LIN {X 0,Y 272.995,Z 1069.366,A -85,B 0,C 180,E1 12162.479,E2 12162.479} C_VEL
LIN {X 0,Y 273.086,Z 1073.952,A -85,B 0,C 180,E1 12158.633,E2 12158.633} C_VEL
LIN {X 0,Y 273.548,Z 1076.686,A -85,B 0,C 180,E1 12155.032,E2 12155.032} C_VEL
LIN {X 0,Y 273.964,Z 1077.76,A -85,B 0,C 180,E1 12151.673,E2 12151.673} C_VEL
LIN {X 0,Y 274.031,Z 1077.444,A -85,B 0,C 180,E1 12148.536,E2 12148.536} C_VEL
LIN {X 0,Y 273.725,Z 1075.691,A -85,B 0,C 180,E1 12145.18,E2 12145.18} C_VEL
LIN {X 0,Y 273.314,Z 1072.175,A -85,B 0,C 180,E1 12141.585,E2 12141.585} C_VEL
LIN {X 0,Y 273.199,Z 1066.916,A -85,B 0,C 180,E1 12137.959,E2 12137.959} C_VEL
LIN {X 0,Y 273.666,Z 1059.821,A -85,B 0,C 180,E1 12134.313,E2 12134.313} C_VEL
LIN {X 0,Y 274.877,Z 1050.701,A -85,B 0,C 180,E1 12130.669,E2 12130.669} C_VEL
LIN {X 0,Y 276.832,Z 1040.026,A -85,B 0,C 180,E1 12127.265,E2 12127.265} C_VEL
LIN {X 0,Y 279.412,Z 1027.805,A -85,B 0,C 180,E1 12124.114,E2 12124.114} C_VEL
LIN {X 0,Y 282.522,Z 1014.014,A -85,B 0,C 180,E1 12121.228,E2 12121.228} C_VEL
LIN {X 0,Y 285.89,Z 999.163,A -85,B 0,C 180,E1 12118.71,E2 12118.71} C_VEL
LIN {X 0,Y 289.318,Z 983.345,A -85,B 0,C 180,E1 12116.549,E2 12116.549} C_VEL
LIN {X 0,Y 292.639,Z 966.616,A -85,B 0,C 180,E1 12114.73,E2 12114.73} C_VEL
LIN {X 0,Y 295.712,Z 948.926,A -85,B 0,C 180,E1 12113.239,E2 12113.239} C_VEL
LIN {X 0,Y 298.36,Z 930.328,A -85,B 0,C 180,E1 12112.082,E2 12112.082} C_VEL
LIN {X 0,Y 300.252,Z 911.657,A -85,B 0,C 180,E1 12111.268,E2 12111.268} C_VEL
LIN {X 0,Y 301.36,Z 889.6,A -85,B 0,C 180,E1 12110.665,E2 12110.665} C_VEL
LIN {X 0,Y 306.573,Z 751.848,A -85,B 0,C 180,E1 12107.521,E2 12107.521} C_VEL
LIN {X 0,Y 305.583,Z 740.205,A -85,B 0,C 180,E1 12106.999,E2 12106.999} C_VEL
LIN {X 0,Y 309.064,Z 717.613,A -85,B 0,C 180,E1 12105.112,E2 12105.112} C_VEL
LIN {X 0,Y 307.717,Z 708.174,A -85,B 0,C 180,E1 12102.748,E2 12102.748} C_VEL
LIN {X 0,Y 307.382,Z 698.126,A -85,B 0,C 180,E1 12099.852,E2 12099.852} C_VEL
LIN {X 0,Y 308.086,Z 690.154,A -85,B 0,C 180,E1 12097.025,E2 12097.025} C_VEL
LIN {X 0,Y 309.031,Z 686.401,A -85,B 0,C 180,E1 12095.504,E2 12095.504} C_VEL
LIN {X 0,Y 308.64,Z 688.001,A -85,B 0,C 180,E1 12091.921,E2 12091.921} C_VEL
LIN {X 0,Y 309.095,Z 689.328,A -85,B 0,C 180,E1 12090.092,E2 12090.092} C_VEL
LIN {X 0,Y 310.043,Z 693.073,A -85,B 0,C 180,E1 12087.462,E2 12087.462} C_VEL
LIN {X 0,Y 311.425,Z 698.192,A -85,B 0,C 180,E1 12084.871,E2 12084.871} C_VEL
LIN {X 0,Y 312.988,Z 704.764,A -85,B 0,C 180,E1 12082.343,E2 12082.343} C_VEL
LIN {X 0,Y 314.593,Z 713.54,A -85,B 0,C 180,E1 12079.688,E2 12079.688} C_VEL
LIN {X 0,Y 315.406,Z 720.749,A -85,B 0,C 180,E1 12077.908,E2 12077.908} C_VEL
LIN {X 0,Y 311.769,Z 746.11,A -85,B 0,C 180,E1 12074.225,E2 12074.225} C_VEL
LIN {X 0,Y 312.167,Z 749.946,A -85,B 0,C 180,E1 12073.919,E2 12073.919} C_VEL
LIN {X 0,Y 302.573,Z 860.757,A -85,B 0,C 180,E1 12070.273,E2 12070.273} C_VEL
LIN {X 0,Y 301.167,Z 887.675,A -85,B 0,C 180,E1 12069.157,E2 12069.157} C_VEL
LIN {X 0,Y 299.803,Z 903.792,A -85,B 0,C 180,E1 12068.148,E2 12068.148} C_VEL
LIN {X 0,Y 297.855,Z 918.992,A -85,B 0,C 180,E1 12066.844,E2 12066.844} C_VEL
LIN {X 0,Y 295.433,Z 933.273,A -85,B 0,C 180,E1 12065.243,E2 12065.243} C_VEL
LIN {X 0,Y 292.379,Z 947.73,A -85,B 0,C 180,E1 12063.136,E2 12063.136} C_VEL
LIN {X 0,Y 289.471,Z 959.226,A -85,B 0,C 180,E1 12060.989,E2 12060.989} C_VEL
LIN {X 0,Y 286.549,Z 969.342,A -85,B 0,C 180,E1 12058.6,E2 12058.6} C_VEL
LIN {X 0,Y 283.732,Z 978.089,A -85,B 0,C 180,E1 12055.958,E2 12055.958} C_VEL
LIN {X 0,Y 281.077,Z 985.57,A -85,B 0,C 180,E1 12052.97,E2 12052.97} C_VEL
LIN {X 0,Y 278.881,Z 991.049,A -85,B 0,C 180,E1 12049.881,E2 12049.881} C_VEL
LIN {X 0,Y 277.157,Z 994.834,A -85,B 0,C 180,E1 12046.65,E2 12046.65} C_VEL
LIN {X 0,Y 275.923,Z 996.716,A -85,B 0,C 180,E1 12043.365,E2 12043.365} C_VEL
LIN {X 0,Y 275.168,Z 996.843,A -85,B 0,C 180,E1 12040.028,E2 12040.028} C_VEL
LIN {X 0,Y 274.817,Z 995.053,A -85,B 0,C 180,E1 12036.635,E2 12036.635} C_VEL
LIN {X 0,Y 274.858,Z 991.649,A -85,B 0,C 180,E1 12033.42,E2 12033.42} C_VEL
LIN {X 0,Y 275.278,Z 986.292,A -85,B 0,C 180,E1 12030.158,E2 12030.158} C_VEL
LIN {X 0,Y 276.066,Z 979.37,A -85,B 0,C 180,E1 12027.093,E2 12027.093} C_VEL
LIN {X 0,Y 277.27,Z 970.164,A -85,B 0,C 180,E1 12023.999,E2 12023.999} C_VEL
LIN {X 0,Y 278.662,Z 960.149,A -85,B 0,C 180,E1 12021.367,E2 12021.367} C_VEL
LIN {X 0,Y 280.353,Z 947.978,A -85,B 0,C 180,E1 12018.81,E2 12018.81} C_VEL
LIN {X 0,Y 282.105,Z 934.37,A -85,B 0,C 180,E1 12016.56,E2 12016.56} C_VEL
LIN {X 0,Y 283.657,Z 920.721,A -85,B 0,C 180,E1 12014.757,E2 12014.757} C_VEL
LIN {X 0,Y 285.152,Z 904.969,A -85,B 0,C 180,E1 12013.138,E2 12013.138} C_VEL
LIN {X 0,Y 286.275,Z 889.331,A -85,B 0,C 180,E1 12011.932,E2 12011.932} C_VEL
LIN {X 0,Y 287.078,Z 871.902,A -85,B 0,C 180,E1 12010.982,E2 12010.982} C_VEL
LIN {X 0,Y 288.495,Z 824.298,A -85,B 0,C 180,E1 12009.46,E2 12009.46} C_VEL
LIN {X 0,Y 292.505,Z 735.615,A -85,B 0,C 180,E1 12006.795,E2 12006.795} C_VEL
LIN {X 0,Y 291.348,Z 726.273,A -85,B 0,C 180,E1 12006.299,E2 12006.299} C_VEL
LIN {X 0,Y 293.227,Z 697.722,A -85,B 0,C 180,E1 12002.258,E2 12002.258} C_VEL
LIN {X 0,Y 288.187,Z 679.048,A -85,B 0,C 180,E1 11998.834,E2 11998.834} C_VEL
LIN {X 0,Y 285.826,Z 671.112,A -85,B 0,C 180,E1 11997.219,E2 11997.219} C_VEL
LIN {X 0,Y 285.73,Z 671.591,A -85,B 0,C 180,E1 11996.832,E2 11996.832} C_VEL
LIN {X 0,Y 289.394,Z 684.621,A -85,B 0,C 180,E1 11992.981,E2 11992.981} C_VEL
LIN {X 0,Y 292.427,Z 697.104,A -85,B 0,C 180,E1 11989.63,E2 11989.63} C_VEL
LIN {X 0,Y 296.094,Z 705.518,A -85,B 0,C 180,E1 11988.815,E2 11988.815} C_VEL
LIN {X 0,Y 302.336,Z 742.558,A -85,B 0,C 180,E1 11986.947,E2 11986.947} C_VEL
LIN {X 0,Y 297.857,Z 856.262,A -85,B 0,C 180,E1 11984.229,E2 11984.229} C_VEL
LIN {X 0,Y 296.8,Z 873.568,A -85,B 0,C 180,E1 11983.479,E2 11983.479} C_VEL
LIN {X 0,Y 295.19,Z 890.075,A -85,B 0,C 180,E1 11982.421,E2 11982.421} C_VEL
LIN {X 0,Y 293.048,Z 906.282,A -85,B 0,C 180,E1 11981.016,E2 11981.016} C_VEL
LIN {X 0,Y 290.554,Z 921.277,A -85,B 0,C 180,E1 11979.308,E2 11979.308} C_VEL
LIN {X 0,Y 287.726,Z 935.883,A -85,B 0,C 180,E1 11977.187,E2 11977.187} C_VEL
LIN {X 0,Y 284.947,Z 948.755,A -85,B 0,C 180,E1 11974.831,E2 11974.831} C_VEL
LIN {X 0,Y 282.29,Z 960.021,A -85,B 0,C 180,E1 11972.233,E2 11972.233} C_VEL
LIN {X 0,Y 279.893,Z 969.883,A -85,B 0,C 180,E1 11969.386,E2 11969.386} C_VEL
LIN {X 0,Y 277.876,Z 978.33,A -85,B 0,C 180,E1 11966.287,E2 11966.287} C_VEL
LIN {X 0,Y 276.311,Z 985.211,A -85,B 0,C 180,E1 11962.933,E2 11962.933} C_VEL
LIN {X 0,Y 275.28,Z 990.531,A -85,B 0,C 180,E1 11959.325,E2 11959.325} C_VEL
LIN {X 0,Y 274.824,Z 993.823,A -85,B 0,C 180,E1 11955.892,E2 11955.892} C_VEL
LIN {X 0,Y 274.806,Z 995.381,A -85,B 0,C 180,E1 11952.798,E2 11952.798} C_VEL
LIN {X 0,Y 273.962,Z 995.9,A -85,B 0,C 180,E1 11951.19,E2 11951.19} C_VEL
LIN {X 0,Y 269.946,Z 996.336,A -85,B 0,C 180,E1 11948.118,E2 11948.118} C_VEL
LIN {X 0,Y 268.383,Z 995.852,A -85,B 0,C 180,E1 11946.127,E2 11946.127} C_VEL
LIN {X 0,Y 268.434,Z 995.457,A -85,B 0,C 180,E1 11945.418,E2 11945.418} C_VEL
LIN {X 0,Y 270.205,Z 992.308,A -85,B 0,C 180,E1 11941.727,E2 11941.727} C_VEL
LIN {X 0,Y 272.718,Z 987.361,A -85,B 0,C 180,E1 11938.134,E2 11938.134} C_VEL
LIN {X 0,Y 275.825,Z 980.766,A -85,B 0,C 180,E1 11934.805,E2 11934.805} C_VEL
LIN {X 0,Y 279.405,Z 972.721,A -85,B 0,C 180,E1 11931.751,E2 11931.751} C_VEL
LIN {X 0,Y 283.302,Z 963.298,A -85,B 0,C 180,E1 11928.971,E2 11928.971} C_VEL
LIN {X 0,Y 287.374,Z 952.502,A -85,B 0,C 180,E1 11926.457,E2 11926.457} C_VEL
LIN {X 0,Y 291.479,Z 940.225,A -85,B 0,C 180,E1 11924.199,E2 11924.199} C_VEL
LIN {X 0,Y 295.51,Z 926.416,A -85,B 0,C 180,E1 11922.185,E2 11922.185} C_VEL
LIN {X 0,Y 299.136,Z 911.731,A -85,B 0,C 180,E1 11920.5,E2 11920.5} C_VEL
LIN {X 0,Y 302.219,Z 896.085,A -85,B 0,C 180,E1 11919.121,E2 11919.121} C_VEL
LIN {X 0,Y 304.672,Z 879.206,A -85,B 0,C 180,E1 11918.018,E2 11918.018} C_VEL
LIN {X 0,Y 306.304,Z 861.93,A -85,B 0,C 180,E1 11917.234,E2 11917.234} C_VEL
LIN {X 0,Y 308.486,Z 821.252,A -85,B 0,C 180,E1 11916.181,E2 11916.181} C_VEL
LIN {X 0,Y 312.469,Z 748.774,A -85,B 0,C 180,E1 11914.471,E2 11914.471} C_VEL
LIN {X 0,Y 308.914,Z 728.999,A -85,B 0,C 180,E1 11913.024,E2 11913.024} C_VEL
LIN {X 0,Y 301.266,Z 715.082,A -85,B 0,C 180,E1 11910.738,E2 11910.738} C_VEL
LIN {X 0,Y 293.815,Z 703.135,A -85,B 0,C 180,E1 11908.286,E2 11908.286} C_VEL
LIN {X 0,Y 291.034,Z 698.461,A -85,B 0,C 180,E1 11907.19,E2 11907.19} C_VEL
LIN {X 0,Y 288.191,Z 689.335,A -85,B 0,C 180,E1 11903.163,E2 11903.163} C_VEL
LIN {X 0,Y 285.796,Z 682.579,A -85,B 0,C 180,E1 11899.625,E2 11899.625} C_VEL
LIN {X 0,Y 283.743,Z 676.858,A -85,B 0,C 180,E1 11896.164,E2 11896.164} C_VEL
LIN {X 0,Y 282.053,Z 672.747,A -85,B 0,C 180,E1 11893.114,E2 11893.114} C_VEL
LIN {X 0,Y 280.668,Z 669.223,A -85,B 0,C 180,E1 11890.053,E2 11890.053} C_VEL
LIN {X 0,Y 279.067,Z 665.356,A -85,B 0,C 180,E1 11885.758,E2 11885.758} C_VEL
LIN {X 0,Y 277.614,Z 661.831,A -85,B 0,C 180,E1 11878.762,E2 11878.762} C_VEL
LIN {X 0,Y 277.53,Z 661.462,A -85,B 0,C 180,E1 11874.211,E2 11874.211} C_VEL
LIN {X 0,Y 277.897,Z 662.139,A -85,B 0,C 180,E1 11870.343,E2 11870.343} C_VEL
LIN {X 0,Y 280.251,Z 666.587,A -85,B 0,C 180,E1 11862.776,E2 11862.776} C_VEL
LIN {X 0,Y 282.567,Z 671.568,A -85,B 0,C 180,E1 11858.19,E2 11858.19} C_VEL
LIN {X 0,Y 284.65,Z 676.264,A -85,B 0,C 180,E1 11854.848,E2 11854.848} C_VEL
LIN {X 0,Y 286.664,Z 680.778,A -85,B 0,C 180,E1 11852.136,E2 11852.136} C_VEL
LIN {X 0,Y 289.552,Z 687.256,A -85,B 0,C 180,E1 11848.804,E2 11848.804} C_VEL
LIN {X 0,Y 293.265,Z 696.674,A -85,B 0,C 180,E1 11844.817,E2 11844.817} C_VEL
LIN {X 0,Y 296.357,Z 704.96,A -85,B 0,C 180,E1 11841.934,E2 11841.934} C_VEL
LIN {X 0,Y 304.493,Z 718.116,A -85,B 0,C 180,E1 11839.384,E2 11839.384} C_VEL
LIN {X 0,Y 311.329,Z 730.667,A -85,B 0,C 180,E1 11837.403,E2 11837.403} C_VEL
LIN {X 0,Y 313.145,Z 757.234,A -85,B 0,C 180,E1 11836.102,E2 11836.102} C_VEL
LIN {X 0,Y 305.231,Z 903.639,A -85,B 0,C 180,E1 11832.685,E2 11832.685} C_VEL
LIN {X 0,Y 303.045,Z 922.451,A -85,B 0,C 180,E1 11831.974,E2 11831.974} C_VEL
LIN {X 0,Y 300.035,Z 939.917,A -85,B 0,C 180,E1 11831.033,E2 11831.033} C_VEL
LIN {X 0,Y 296.257,Z 957.297,A -85,B 0,C 180,E1 11829.758,E2 11829.758} C_VEL
LIN {X 0,Y 291.833,Z 974.657,A -85,B 0,C 180,E1 11828.075,E2 11828.075} C_VEL
LIN {X 0,Y 287.145,Z 990.928,A -85,B 0,C 180,E1 11826.048,E2 11826.048} C_VEL
LIN {X 0,Y 282.513,Z 1005.741,A -85,B 0,C 180,E1 11823.726,E2 11823.726} C_VEL
LIN {X 0,Y 277.892,Z 1019.902,A -85,B 0,C 180,E1 11820.965,E2 11820.965} C_VEL
LIN {X 0,Y 273.727,Z 1032.637,A -85,B 0,C 180,E1 11817.875,E2 11817.875} C_VEL
LIN {X 0,Y 270.199,Z 1043.975,A -85,B 0,C 180,E1 11814.452,E2 11814.452} C_VEL
LIN {X 0,Y 267.526,Z 1053.664,A -85,B 0,C 180,E1 11810.796,E2 11810.796} C_VEL
LIN {X 0,Y 265.79,Z 1061.928,A -85,B 0,C 180,E1 11806.837,E2 11806.837} C_VEL
LIN {X 0,Y 265.04,Z 1068.271,A -85,B 0,C 180,E1 11802.86,E2 11802.86} C_VEL
LIN {X 0,Y 265.11,Z 1072.865,A -85,B 0,C 180,E1 11798.838,E2 11798.838} C_VEL
LIN {X 0,Y 265.587,Z 1075.513,A -85,B 0,C 180,E1 11795.183,E2 11795.183} C_VEL
LIN {X 0,Y 266.044,Z 1076.575,A -85,B 0,C 180,E1 11791.722,E2 11791.722} C_VEL
LIN {X 0,Y 266.121,Z 1076.205,A -85,B 0,C 180,E1 11788.492,E2 11788.492} C_VEL
LIN {X 0,Y 265.786,Z 1074.385,A -85,B 0,C 180,E1 11785.036,E2 11785.036} C_VEL
LIN {X 0,Y 265.354,Z 1070.79,A -85,B 0,C 180,E1 11781.331,E2 11781.331} C_VEL
LIN {X 0,Y 265.258,Z 1065.444,A -85,B 0,C 180,E1 11777.592,E2 11777.592} C_VEL
LIN {X 0,Y 265.794,Z 1058.252,A -85,B 0,C 180,E1 11773.836,E2 11773.836} C_VEL
LIN {X 0,Y 267.02,Z 1049.627,A -85,B 0,C 180,E1 11770.305,E2 11770.305} C_VEL
LIN {X 0,Y 269.075,Z 1038.942,A -85,B 0,C 180,E1 11766.803,E2 11766.803} C_VEL
LIN {X 0,Y 271.781,Z 1026.722,A -85,B 0,C 180,E1 11763.566,E2 11763.566} C_VEL
LIN {X 0,Y 275.034,Z 1012.929,A -85,B 0,C 180,E1 11760.607,E2 11760.607} C_VEL
LIN {X 0,Y 278.545,Z 998.068,A -85,B 0,C 180,E1 11758.03,E2 11758.03} C_VEL
LIN {X 0,Y 282.111,Z 982.224,A -85,B 0,C 180,E1 11755.822,E2 11755.822} C_VEL
LIN {X 0,Y 285.56,Z 965.436,A -85,B 0,C 180,E1 11753.967,E2 11753.967} C_VEL
LIN {X 0,Y 288.748,Z 947.603,A -85,B 0,C 180,E1 11752.45,E2 11752.45} C_VEL
LIN {X 0,Y 291.428,Z 929.253,A -85,B 0,C 180,E1 11751.296,E2 11751.296} C_VEL
LIN {X 0,Y 293.355,Z 910.609,A -85,B 0,C 180,E1 11750.475,E2 11750.475} C_VEL
LIN {X 0,Y 294.515,Z 887.782,A -85,B 0,C 180,E1 11749.847,E2 11749.847} C_VEL
LIN {X 0,Y 300.007,Z 753.248,A -85,B 0,C 180,E1 11746.699,E2 11746.699} C_VEL
LIN {X 0,Y 304.477,Z 724.953,A -85,B 0,C 180,E1 11744.284,E2 11744.284} C_VEL
LIN {X 0,Y 305.072,Z 721.863,A -85,B 0,C 180,E1 11744.012,E2 11744.012} C_VEL
LIN {X 0,Y 304.024,Z 710.117,A -85,B 0,C 180,E1 11740.85,E2 11740.85} C_VEL
LIN {X 0,Y 304.177,Z 703.703,A -85,B 0,C 180,E1 11738.89,E2 11738.89} C_VEL
LIN {X 0,Y 305.114,Z 696.484,A -85,B 0,C 180,E1 11736.278,E2 11736.278} C_VEL
LIN {X 0,Y 305.869,Z 693.866,A -85,B 0,C 180,E1 11735.122,E2 11735.122} C_VEL
LIN {X 0,Y 305.772,Z 696.105,A -85,B 0,C 180,E1 11730.617,E2 11730.617} C_VEL
LIN {X 0,Y 306.432,Z 700.334,A -85,B 0,C 180,E1 11727.602,E2 11727.602} C_VEL
LIN {X 0,Y 307.59,Z 705.375,A -85,B 0,C 180,E1 11724.997,E2 11724.997} C_VEL
LIN {X 0,Y 308.982,Z 712.642,A -85,B 0,C 180,E1 11722.247,E2 11722.247} C_VEL
LIN {X 0,Y 310.084,Z 720.981,A -85,B 0,C 180,E1 11719.789,E2 11719.789} C_VEL
LIN {X 0,Y 310.417,Z 725.229,A -85,B 0,C 180,E1 11718.739,E2 11718.739} C_VEL
LIN {X 0,Y 306.869,Z 747.846,A -85,B 0,C 180,E1 11715.411,E2 11715.411} C_VEL
LIN {X 0,Y 307.246,Z 752.01,A -85,B 0,C 180,E1 11715.054,E2 11715.054} C_VEL
LIN {X 0,Y 296.996,Z 861.826,A -85,B 0,C 180,E1 11711.352,E2 11711.352} C_VEL
LIN {X 0,Y 295.444,Z 889.256,A -85,B 0,C 180,E1 11710.191,E2 11710.191} C_VEL
LIN {X 0,Y 293.861,Z 906.037,A -85,B 0,C 180,E1 11709.103,E2 11709.103} C_VEL
LIN {X 0,Y 291.746,Z 920.887,A -85,B 0,C 180,E1 11707.78,E2 11707.78} C_VEL
LIN {X 0,Y 289.169,Z 935.064,A -85,B 0,C 180,E1 11706.153,E2 11706.153} C_VEL
LIN {X 0,Y 286.048,Z 948.797,A -85,B 0,C 180,E1 11704.109,E2 11704.109} C_VEL
LIN {X 0,Y 283.063,Z 959.845,A -85,B 0,C 180,E1 11702.024,E2 11702.024} C_VEL
LIN {X 0,Y 279.677,Z 970.898,A -85,B 0,C 180,E1 11699.385,E2 11699.385} C_VEL
LIN {X 0,Y 276.64,Z 979.558,A -85,B 0,C 180,E1 11696.684,E2 11696.684} C_VEL
LIN {X 0,Y 273.704,Z 987.181,A -85,B 0,C 180,E1 11693.538,E2 11693.538} C_VEL
LIN {X 0,Y 271.256,Z 992.774,A -85,B 0,C 180,E1 11690.237,E2 11690.237} C_VEL
LIN {X 0,Y 269.513,Z 996.196,A -85,B 0,C 180,E1 11687.138,E2 11687.138} C_VEL
LIN {X 0,Y 268.155,Z 998.055,A -85,B 0,C 180,E1 11683.76,E2 11683.76} C_VEL
LIN {X 0,Y 267.312,Z 998.154,A -85,B 0,C 180,E1 11680.327,E2 11680.327} C_VEL
LIN {X 0,Y 266.903,Z 996.337,A -85,B 0,C 180,E1 11676.837,E2 11676.837} C_VEL
LIN {X 0,Y 266.92,Z 992.916,A -85,B 0,C 180,E1 11673.527,E2 11673.527} C_VEL
LIN {X 0,Y 267.333,Z 987.523,A -85,B 0,C 180,E1 11670.169,E2 11670.169} C_VEL
LIN {X 0,Y 268.133,Z 980.573,A -85,B 0,C 180,E1 11667.014,E2 11667.014} C_VEL
LIN {X 0,Y 269.371,Z 971.321,A -85,B 0,C 180,E1 11663.83,E2 11663.83} C_VEL
LIN {X 0,Y 270.881,Z 960.748,A -85,B 0,C 180,E1 11660.998,E2 11660.998} C_VEL
LIN {X 0,Y 272.617,Z 948.578,A -85,B 0,C 180,E1 11658.406,E2 11658.406} C_VEL
LIN {X 0,Y 274.477,Z 934.593,A -85,B 0,C 180,E1 11656.056,E2 11656.056} C_VEL
LIN {X 0,Y 276.106,Z 920.533,A -85,B 0,C 180,E1 11654.191,E2 11654.191} C_VEL
LIN {X 0,Y 277.578,Z 905.504,A -85,B 0,C 180,E1 11652.625,E2 11652.625} C_VEL
LIN {X 0,Y 278.775,Z 889.169,A -85,B 0,C 180,E1 11651.356,E2 11651.356} C_VEL
LIN {X 0,Y 279.565,Z 872.233,A -85,B 0,C 180,E1 11650.43,E2 11650.43} C_VEL
LIN {X 0,Y 281.098,Z 824.122,A -85,B 0,C 180,E1 11648.845,E2 11648.845} C_VEL
LIN {X 0,Y 285.233,Z 736.528,A -85,B 0,C 180,E1 11646.135,E2 11646.135} C_VEL
LIN {X 0,Y 284.099,Z 727.688,A -85,B 0,C 180,E1 11645.685,E2 11645.685} C_VEL
LIN {X 0,Y 285.945,Z 700.168,A -85,B 0,C 180,E1 11641.753,E2 11641.753} C_VEL
LIN {X 0,Y 281.051,Z 681.958,A -85,B 0,C 180,E1 11638.356,E2 11638.356} C_VEL
LIN {X 0,Y 279.384,Z 676.226,A -85,B 0,C 180,E1 11637.149,E2 11637.149} C_VEL
LIN {X 0,Y 279.291,Z 676.82,A -85,B 0,C 180,E1 11636.699,E2 11636.699} C_VEL
LIN {X 0,Y 283.041,Z 690.731,A -85,B 0,C 180,E1 11632.538,E2 11632.538} C_VEL
LIN {X 0,Y 284.718,Z 697.599,A -85,B 0,C 180,E1 11630.706,E2 11630.706} C_VEL
LIN {X 0,Y 289.858,Z 708.653,A -85,B 0,C 180,E1 11629.597,E2 11629.597} C_VEL
LIN {X 0,Y 295.639,Z 743.871,A -85,B 0,C 180,E1 11627.772,E2 11627.772} C_VEL
LIN {X 0,Y 290.996,Z 856.789,A -85,B 0,C 180,E1 11625.023,E2 11625.023} C_VEL
LIN {X 0,Y 289.911,Z 874.011,A -85,B 0,C 180,E1 11624.269,E2 11624.269} C_VEL
LIN {X 0,Y 288.15,Z 891.3,A -85,B 0,C 180,E1 11623.138,E2 11623.138} C_VEL
LIN {X 0,Y 285.919,Z 907.424,A -85,B 0,C 180,E1 11621.703,E2 11621.703} C_VEL
LIN {X 0,Y 283.323,Z 922.364,A -85,B 0,C 180,E1 11619.958,E2 11619.958} C_VEL
LIN {X 0,Y 280.379,Z 936.953,A -85,B 0,C 180,E1 11617.789,E2 11617.789} C_VEL
LIN {X 0,Y 277.481,Z 949.814,A -85,B 0,C 180,E1 11615.376,E2 11615.376} C_VEL
LIN {X 0,Y 274.711,Z 961.081,A -85,B 0,C 180,E1 11612.713,E2 11612.713} C_VEL
LIN {X 0,Y 272.207,Z 970.951,A -85,B 0,C 180,E1 11609.79,E2 11609.79} C_VEL
LIN {X 0,Y 270.096,Z 979.412,A -85,B 0,C 180,E1 11606.605,E2 11606.605} C_VEL
LIN {X 0,Y 268.458,Z 986.314,A -85,B 0,C 180,E1 11603.156,E2 11603.156} C_VEL
LIN {X 0,Y 267.379,Z 991.656,A -85,B 0,C 180,E1 11599.442,E2 11599.442} C_VEL
LIN {X 0,Y 266.904,Z 994.974,A -85,B 0,C 180,E1 11595.907,E2 11595.907} C_VEL
LIN {X 0,Y 266.934,Z 996.705,A -85,B 0,C 180,E1 11592.113,E2 11592.113} C_VEL
LIN {X 0,Y 267.545,Z 996.672,A -85,B 0,C 180,E1 11588.286,E2 11588.286} C_VEL
LIN {X 0,Y 268.434,Z 995.457,A -85,B 0,C 180,E1 11585.418,E2 11585.418} C_VEL
LIN {X 0,Y 268.139,Z 994.48,A -85,B 0,C 180,E1 11583.775,E2 11583.775} C_VEL
LIN {X 0,Y 264.884,Z 991.769,A -85,B 0,C 180,E1 11580.034,E2 11580.034} C_VEL
LIN {X 0,Y 264.691,Z 989.716,A -85,B 0,C 180,E1 11578.285,E2 11578.285} C_VEL
LIN {X 0,Y 264.919,Z 989.214,A -85,B 0,C 180,E1 11577.943,E2 11577.943} C_VEL
LIN {X 0,Y 268.222,Z 982.735,A -85,B 0,C 180,E1 11574.443,E2 11574.443} C_VEL
LIN {X 0,Y 272.121,Z 974.468,A -85,B 0,C 180,E1 11571.166,E2 11571.166} C_VEL
LIN {X 0,Y 276.428,Z 964.619,A -85,B 0,C 180,E1 11568.17,E2 11568.17} C_VEL
LIN {X 0,Y 280.69,Z 953.932,A -85,B 0,C 180,E1 11565.617,E2 11565.617} C_VEL
LIN {X 0,Y 285.043,Z 941.599,A -85,B 0,C 180,E1 11563.294,E2 11563.294} C_VEL
LIN {X 0,Y 289.279,Z 927.807,A -85,B 0,C 180,E1 11561.24,E2 11561.24} C_VEL
LIN {X 0,Y 293.034,Z 913.325,A -85,B 0,C 180,E1 11559.545,E2 11559.545} C_VEL
LIN {X 0,Y 296.291,Z 897.764,A -85,B 0,C 180,E1 11558.138,E2 11558.138} C_VEL
LIN {X 0,Y 298.872,Z 881.007,A -85,B 0,C 180,E1 11557.014,E2 11557.014} C_VEL
LIN {X 0,Y 300.641,Z 863.495,A -85,B 0,C 180,E1 11556.195,E2 11556.195} C_VEL
LIN {X 0,Y 302.405,Z 831.917,A -85,B 0,C 180,E1 11555.337,E2 11555.337} C_VEL
LIN {X 0,Y 307.08,Z 750.315,A -85,B 0,C 180,E1 11553.386,E2 11553.386} C_VEL
LIN {X 0,Y 304.096,Z 733.373,A -85,B 0,C 180,E1 11552.102,E2 11552.102} C_VEL
LIN {X 0,Y 297.245,Z 720.673,A -85,B 0,C 180,E1 11549.941,E2 11549.941} C_VEL
LIN {X 0,Y 290.393,Z 709.436,A -85,B 0,C 180,E1 11547.588,E2 11547.588} C_VEL
LIN {X 0,Y 285.777,Z 702.516,A -85,B 0,C 180,E1 11545.879,E2 11545.879} C_VEL
LIN {X 0,Y 283.743,Z 699.193,A -85,B 0,C 180,E1 11545.016,E2 11545.016} C_VEL
LIN {X 0,Y 281.298,Z 691.703,A -85,B 0,C 180,E1 11541.476,E2 11541.476} C_VEL
LIN {X 0,Y 279.014,Z 685.186,A -85,B 0,C 180,E1 11537.735,E2 11537.735} C_VEL
LIN {X 0,Y 277.542,Z 681.234,A -85,B 0,C 180,E1 11535.034,E2 11535.034} C_VEL
LIN {X 0,Y 276.417,Z 678.263,A -85,B 0,C 180,E1 11532.748,E2 11532.748} C_VEL
LIN {X 0,Y 275.166,Z 674.971,A -85,B 0,C 180,E1 11529.834,E2 11529.834} C_VEL
LIN {X 0,Y 273.758,Z 671.326,A -85,B 0,C 180,E1 11525.66,E2 11525.66} C_VEL
LIN {X 0,Y 272.448,Z 667.886,A -85,B 0,C 180,E1 11518.528,E2 11518.528} C_VEL
LIN {X 0,Y 272.438,Z 667.623,A -85,B 0,C 180,E1 11513.679,E2 11513.679} C_VEL
LIN {X 0,Y 272.818,Z 668.418,A -85,B 0,C 180,E1 11510.082,E2 11510.082} C_VEL
LIN {X 0,Y 275.057,Z 672.683,A -85,B 0,C 180,E1 11502.876,E2 11502.876} C_VEL
LIN {X 0,Y 277.317,Z 677.745,A -85,B 0,C 180,E1 11498.201,E2 11498.201} C_VEL
LIN {X 0,Y 279.269,Z 682.155,A -85,B 0,C 180,E1 11495.01,E2 11495.01} C_VEL
LIN {X 0,Y 281.237,Z 686.689,A -85,B 0,C 180,E1 11492.243,E2 11492.243} C_VEL
LIN {X 0,Y 283.926,Z 692.814,A -85,B 0,C 180,E1 11489.06,E2 11489.06} C_VEL
LIN {X 0,Y 287.559,Z 702.277,A -85,B 0,C 180,E1 11484.991,E2 11484.991} C_VEL
LIN {X 0,Y 288.877,Z 705.256,A -85,B 0,C 180,E1 11484.018,E2 11484.018} C_VEL
LIN {X 0,Y 296.981,Z 717.914,A -85,B 0,C 180,E1 11481.229,E2 11481.229} C_VEL
LIN {X 0,Y 304.225,Z 730.679,A -85,B 0,C 180,E1 11478.967,E2 11478.967} C_VEL
LIN {X 0,Y 306.295,Z 735.066,A -85,B 0,C 180,E1 11478.333,E2 11478.333} C_VEL
LIN {X 0,Y 307.711,Z 758.585,A -85,B 0,C 180,E1 11477.171,E2 11477.171} C_VEL
LIN {X 0,Y 299.54,Z 902.9,A -85,B 0,C 180,E1 11473.764,E2 11473.764} C_VEL
LIN {X 0,Y 297.28,Z 921.628,A -85,B 0,C 180,E1 11473.048,E2 11473.048} C_VEL
LIN {X 0,Y 294.028,Z 939.702,A -85,B 0,C 180,E1 11472.06,E2 11472.06} C_VEL
LIN {X 0,Y 290.11,Z 956.924,A -85,B 0,C 180,E1 11470.776,E2 11470.776} C_VEL
LIN {X 0,Y 285.506,Z 974.167,A -85,B 0,C 180,E1 11469.077,E2 11469.077} C_VEL
LIN {X 0,Y 280.747,Z 989.921,A -85,B 0,C 180,E1 11467.084,E2 11467.084} C_VEL
LIN {X 0,Y 275.804,Z 1004.93,A -85,B 0,C 180,E1 11464.691,E2 11464.691} C_VEL
LIN {X 0,Y 271.071,Z 1018.621,A -85,B 0,C 180,E1 11461.966,E2 11461.966} C_VEL
LIN {X 0,Y 266.485,Z 1031.785,A -85,B 0,C 180,E1 11458.702,E2 11458.702} C_VEL
LIN {X 0,Y 262.75,Z 1042.963,A -85,B 0,C 180,E1 11455.226,E2 11455.226} C_VEL
LIN {X 0,Y 259.785,Z 1052.886,A -85,B 0,C 180,E1 11451.345,E2 11451.345} C_VEL
LIN {X 0,Y 257.943,Z 1060.88,A -85,B 0,C 180,E1 11447.365,E2 11447.365} C_VEL
LIN {X 0,Y 257.091,Z 1067.181,A -85,B 0,C 180,E1 11443.265,E2 11443.265} C_VEL
LIN {X 0,Y 257.123,Z 1071.685,A -85,B 0,C 180,E1 11439.173,E2 11439.173} C_VEL
LIN {X 0,Y 257.625,Z 1074.342,A -85,B 0,C 180,E1 11435.344,E2 11435.344} C_VEL
LIN {X 0,Y 258.123,Z 1075.39,A -85,B 0,C 180,E1 11431.775,E2 11431.775} C_VEL
LIN {X 0,Y 258.222,Z 1075.035,A -85,B 0,C 180,E1 11428.668,E2 11428.668} C_VEL
LIN {X 0,Y 257.88,Z 1073.298,A -85,B 0,C 180,E1 11425.165,E2 11425.165} C_VEL
LIN {X 0,Y 257.428,Z 1069.957,A -85,B 0,C 180,E1 11421.512,E2 11421.512} C_VEL
LIN {X 0,Y 257.296,Z 1064.711,A -85,B 0,C 180,E1 11417.658,E2 11417.658} C_VEL
LIN {X 0,Y 257.82,Z 1057.65,A -85,B 0,C 180,E1 11413.785,E2 11413.785} C_VEL
LIN {X 0,Y 259.17,Z 1048.538,A -85,B 0,C 180,E1 11409.918,E2 11409.918} C_VEL
LIN {X 0,Y 261.334,Z 1037.858,A -85,B 0,C 180,E1 11406.313,E2 11406.313} C_VEL
LIN {X 0,Y 264.176,Z 1025.639,A -85,B 0,C 180,E1 11402.987,E2 11402.987} C_VEL
LIN {X 0,Y 267.58,Z 1011.821,A -85,B 0,C 180,E1 11399.952,E2 11399.952} C_VEL
LIN {X 0,Y 271.084,Z 997.564,A -85,B 0,C 180,E1 11397.417,E2 11397.417} C_VEL
LIN {X 0,Y 274.772,Z 981.802,A -85,B 0,C 180,E1 11395.158,E2 11395.158} C_VEL
LIN {X 0,Y 278.337,Z 965.132,A -85,B 0,C 180,E1 11393.264,E2 11393.264} C_VEL
LIN {X 0,Y 281.647,Z 947.406,A -85,B 0,C 180,E1 11391.708,E2 11391.708} C_VEL
LIN {X 0,Y 284.469,Z 928.8,A -85,B 0,C 180,E1 11390.508,E2 11390.508} C_VEL
LIN {X 0,Y 286.465,Z 910.156,A -85,B 0,C 180,E1 11389.665,E2 11389.665} C_VEL
LIN {X 0,Y 287.647,Z 888.177,A -85,B 0,C 180,E1 11389.042,E2 11389.042} C_VEL
LIN {X 0,Y 292.811,Z 769.055,A -85,B 0,C 180,E1 11386.206,E2 11386.206} C_VEL
LIN {X 0,Y 296.025,Z 754.614,A -85,B 0,C 180,E1 11385.368,E2 11385.368} C_VEL
LIN {X 0,Y 300.936,Z 727.86,A -85,B 0,C 180,E1 11383.033,E2 11383.033} C_VEL
LIN {X 0,Y 301.274,Z 726.134,A -85,B 0,C 180,E1 11382.87,E2 11382.87} C_VEL
LIN {X 0,Y 300.94,Z 712.077,A -85,B 0,C 180,E1 11378.898,E2 11378.898} C_VEL
LIN {X 0,Y 302.088,Z 703.515,A -85,B 0,C 180,E1 11375.814,E2 11375.814} C_VEL
LIN {X 0,Y 302.728,Z 701.344,A -85,B 0,C 180,E1 11374.847,E2 11374.847} C_VEL
LIN {X 0,Y 302.452,Z 703.481,A -85,B 0,C 180,E1 11370.736,E2 11370.736} C_VEL
LIN {X 0,Y 302.874,Z 707.257,A -85,B 0,C 180,E1 11367.955,E2 11367.955} C_VEL
LIN {X 0,Y 303.687,Z 711.722,A -85,B 0,C 180,E1 11365.55,E2 11365.55} C_VEL
LIN {X 0,Y 304.707,Z 718.808,A -85,B 0,C 180,E1 11362.768,E2 11362.768} C_VEL
LIN {X 0,Y 305.493,Z 727.027,A -85,B 0,C 180,E1 11360.299,E2 11360.299} C_VEL
LIN {X 0,Y 305.584,Z 729.853,A -85,B 0,C 180,E1 11359.595,E2 11359.595} C_VEL
LIN {X 0,Y 302.191,Z 749.679,A -85,B 0,C 180,E1 11356.643,E2 11356.643} C_VEL
LIN {X 0,Y 302.529,Z 754.134,A -85,B 0,C 180,E1 11356.235,E2 11356.235} C_VEL
LIN {X 0,Y 291.672,Z 862.886,A -85,B 0,C 180,E1 11352.497,E2 11352.497} C_VEL
LIN {X 0,Y 289.903,Z 890.684,A -85,B 0,C 180,E1 11351.287,E2 11351.287} C_VEL
LIN {X 0,Y 288.189,Z 907.194,A -85,B 0,C 180,E1 11350.191,E2 11350.191} C_VEL
LIN {X 0,Y 285.952,Z 922.142,A -85,B 0,C 180,E1 11348.85,E2 11348.85} C_VEL
LIN {X 0,Y 283.201,Z 936.219,A -85,B 0,C 180,E1 11347.208,E2 11347.208} C_VEL
LIN {X 0,Y 279.99,Z 949.348,A -85,B 0,C 180,E1 11345.228,E2 11345.228} C_VEL
LIN {X 0,Y 276.808,Z 960.633,A -85,B 0,C 180,E1 11343.105,E2 11343.105} C_VEL
LIN {X 0,Y 273.398,Z 970.949,A -85,B 0,C 180,E1 11340.628,E2 11340.628} C_VEL
LIN {X 0,Y 270.097,Z 979.933,A -85,B 0,C 180,E1 11337.878,E2 11337.878} C_VEL
LIN {X 0,Y 267.001,Z 987.385,A -85,B 0,C 180,E1 11334.843,E2 11334.843} C_VEL
LIN {X 0,Y 264.436,Z 992.952,A -85,B 0,C 180,E1 11331.739,E2 11331.739} C_VEL
LIN {X 0,Y 262.259,Z 996.984,A -85,B 0,C 180,E1 11328.342,E2 11328.342} C_VEL
LIN {X 0,Y 260.662,Z 999.21,A -85,B 0,C 180,E1 11324.88,E2 11324.88} C_VEL
LIN {X 0,Y 259.605,Z 999.574,A -85,B 0,C 180,E1 11321.347,E2 11321.347} C_VEL
LIN {X 0,Y 259.057,Z 998.154,A -85,B 0,C 180,E1 11317.775,E2 11317.775} C_VEL
LIN {X 0,Y 258.955,Z 994.72,A -85,B 0,C 180,E1 11314.113,E2 11314.113} C_VEL
LIN {X 0,Y 259.261,Z 990.086,A -85,B 0,C 180,E1 11310.926,E2 11310.926} C_VEL
LIN {X 0,Y 260.044,Z 982.961,A -85,B 0,C 180,E1 11307.432,E2 11307.432} C_VEL
LIN {X 0,Y 261.134,Z 974.844,A -85,B 0,C 180,E1 11304.408,E2 11304.408} C_VEL
LIN {X 0,Y 262.66,Z 964.405,A -85,B 0,C 180,E1 11301.369,E2 11301.369} C_VEL
LIN {X 0,Y 264.367,Z 952.784,A -85,B 0,C 180,E1 11298.701,E2 11298.701} C_VEL
LIN {X 0,Y 266.224,Z 939.627,A -85,B 0,C 180,E1 11296.286,E2 11296.286} C_VEL
LIN {X 0,Y 268.099,Z 924.576,A -85,B 0,C 180,E1 11294.117,E2 11294.117} C_VEL
LIN {X 0,Y 269.679,Z 909.566,A -85,B 0,C 180,E1 11292.438,E2 11292.438} C_VEL
LIN {X 0,Y 271.006,Z 893.269,A -85,B 0,C 180,E1 11291.051,E2 11291.051} C_VEL
LIN {X 0,Y 271.975,Z 874.901,A -85,B 0,C 180,E1 11289.965,E2 11289.965} C_VEL
LIN {X 0,Y 273.209,Z 834.078,A -85,B 0,C 180,E1 11288.544,E2 11288.544} C_VEL
LIN {X 0,Y 277.991,Z 737.548,A -85,B 0,C 180,E1 11285.457,E2 11285.457} C_VEL
LIN {X 0,Y 276.9,Z 728.312,A -85,B 0,C 180,E1 11284.947,E2 11284.947} C_VEL
LIN {X 0,Y 278.704,Z 702.66,A -85,B 0,C 180,E1 11281.226,E2 11281.226} C_VEL
LIN {X 0,Y 273.806,Z 684.386,A -85,B 0,C 180,E1 11277.749,E2 11277.749} C_VEL
LIN {X 0,Y 272.94,Z 681.337,A -85,B 0,C 180,E1 11277.073,E2 11277.073} C_VEL
LIN {X 0,Y 272.733,Z 681.721,A -85,B 0,C 180,E1 11276.686,E2 11276.686} C_VEL
LIN {X 0,Y 276.054,Z 694.408,A -85,B 0,C 180,E1 11272.803,E2 11272.803} C_VEL
LIN {X 0,Y 276.915,Z 697.848,A -85,B 0,C 180,E1 11271.916,E2 11271.916} C_VEL
LIN {X 0,Y 283.701,Z 711.978,A -85,B 0,C 180,E1 11270.402,E2 11270.402} C_VEL
LIN {X 0,Y 288.993,Z 745.134,A -85,B 0,C 180,E1 11268.633,E2 11268.633} C_VEL
LIN {X 0,Y 284.191,Z 857.24,A -85,B 0,C 180,E1 11265.856,E2 11265.856} C_VEL
LIN {X 0,Y 283.062,Z 874.587,A -85,B 0,C 180,E1 11265.088,E2 11265.088} C_VEL
LIN {X 0,Y 281.281,Z 891.502,A -85,B 0,C 180,E1 11263.968,E2 11263.968} C_VEL
LIN {X 0,Y 278.985,Z 907.586,A -85,B 0,C 180,E1 11262.523,E2 11262.523} C_VEL
LIN {X 0,Y 276.28,Z 922.722,A -85,B 0,C 180,E1 11260.742,E2 11260.742} C_VEL
LIN {X 0,Y 273.329,Z 936.813,A -85,B 0,C 180,E1 11258.626,E2 11258.626} C_VEL
LIN {X 0,Y 270.28,Z 949.893,A -85,B 0,C 180,E1 11256.159,E2 11256.159} C_VEL
LIN {X 0,Y 267.359,Z 961.369,A -85,B 0,C 180,E1 11253.431,E2 11253.431} C_VEL
LIN {X 0,Y 264.704,Z 971.38,A -85,B 0,C 180,E1 11250.433,E2 11250.433} C_VEL
LIN {X 0,Y 262.451,Z 979.973,A -85,B 0,C 180,E1 11247.162,E2 11247.162} C_VEL
LIN {X 0,Y 260.79,Z 986.685,A -85,B 0,C 180,E1 11243.838,E2 11243.838} C_VEL
LIN {X 0,Y 259.632,Z 991.979,A -85,B 0,C 180,E1 11240.245,E2 11240.245} C_VEL
LIN {X 0,Y 259.016,Z 995.772,A -85,B 0,C 180,E1 11236.381,E2 11236.381} C_VEL
LIN {X 0,Y 258.996,Z 997.802,A -85,B 0,C 180,E1 11232.47,E2 11232.47} C_VEL
LIN {X 0,Y 259.574,Z 997.996,A -85,B 0,C 180,E1 11228.536,E2 11228.536} C_VEL
LIN {X 0,Y 260.858,Z 996.391,A -85,B 0,C 180,E1 11224.578,E2 11224.578} C_VEL
LIN {X 0,Y 262.811,Z 993.142,A -85,B 0,C 180,E1 11220.859,E2 11220.859} C_VEL
LIN {X 0,Y 264.919,Z 989.214,A -85,B 0,C 180,E1 11217.943,E2 11217.943} C_VEL
LIN {X 0,Y 265.352,Z 986.91,A -85,B 0,C 180,E1 11216.341,E2 11216.341} C_VEL
LIN {X 0,Y 263.829,Z 981.629,A -85,B 0,C 180,E1 11212.905,E2 11212.905} C_VEL
LIN {X 0,Y 264.172,Z 977.892,A -85,B 0,C 180,E1 11211.157,E2 11211.157} C_VEL
LIN {X 0,Y 264.608,Z 976.8,A -85,B 0,C 180,E1 11210.749,E2 11210.749} C_VEL
LIN {X 0,Y 269.032,Z 967.29,A -85,B 0,C 180,E1 11207.697,E2 11207.697} C_VEL
LIN {X 0,Y 273.788,Z 956.063,A -85,B 0,C 180,E1 11204.889,E2 11204.889} C_VEL
LIN {X 0,Y 278.465,Z 943.65,A -85,B 0,C 180,E1 11202.457,E2 11202.457} C_VEL
LIN {X 0,Y 282.853,Z 930.132,A -85,B 0,C 180,E1 11200.38,E2 11200.38} C_VEL
LIN {X 0,Y 286.914,Z 915.329,A -85,B 0,C 180,E1 11198.594,E2 11198.594} C_VEL
LIN {X 0,Y 290.378,Z 899.783,A -85,B 0,C 180,E1 11197.144,E2 11197.144} C_VEL
LIN {X 0,Y 293.115,Z 883.221,A -85,B 0,C 180,E1 11195.994,E2 11195.994} C_VEL
LIN {X 0,Y 295.029,Z 865.666,A -85,B 0,C 180,E1 11195.141,E2 11195.141} C_VEL
LIN {X 0,Y 296.499,Z 840.786,A -85,B 0,C 180,E1 11194.414,E2 11194.414} C_VEL
LIN {X 0,Y 301.839,Z 752.089,A -85,B 0,C 180,E1 11192.279,E2 11192.279} C_VEL
LIN {X 0,Y 299.428,Z 737.842,A -85,B 0,C 180,E1 11191.171,E2 11191.171} C_VEL
LIN {X 0,Y 292.851,Z 725.514,A -85,B 0,C 180,E1 11188.973,E2 11188.973} C_VEL
LIN {X 0,Y 286.779,Z 715.375,A -85,B 0,C 180,E1 11186.785,E2 11186.785} C_VEL
LIN {X 0,Y 280.739,Z 705.969,A -85,B 0,C 180,E1 11184.403,E2 11184.403} C_VEL
LIN {X 0,Y 276.218,Z 699.276,A -85,B 0,C 180,E1 11182.339,E2 11182.339} C_VEL
LIN {X 0,Y 273.898,Z 692.293,A -85,B 0,C 180,E1 11178.518,E2 11178.518} C_VEL
LIN {X 0,Y 272.103,Z 687.26,A -85,B 0,C 180,E1 11175.124,E2 11175.124} C_VEL
LIN {X 0,Y 270.909,Z 684.009,A -85,B 0,C 180,E1 11172.578,E2 11172.578} C_VEL
LIN {X 0,Y 269.801,Z 680.914,A -85,B 0,C 180,E1 11169.816,E2 11169.816} C_VEL
LIN {X 0,Y 268.489,Z 677.33,A -85,B 0,C 180,E1 11165.557,E2 11165.557} C_VEL
LIN {X 0,Y 267.286,Z 674.001,A -85,B 0,C 180,E1 11158.5,E2 11158.5} C_VEL
LIN {X 0,Y 267.296,Z 673.751,A -85,B 0,C 180,E1 11153.557,E2 11153.557} C_VEL
LIN {X 0,Y 267.7,Z 674.574,A -85,B 0,C 180,E1 11150.107,E2 11150.107} C_VEL
LIN {X 0,Y 269.901,Z 678.887,A -85,B 0,C 180,E1 11142.894,E2 11142.894} C_VEL
LIN {X 0,Y 272.005,Z 683.625,A -85,B 0,C 180,E1 11138.433,E2 11138.433} C_VEL
LIN {X 0,Y 273.891,Z 688.047,A -85,B 0,C 180,E1 11135.177,E2 11135.177} C_VEL
LIN {X 0,Y 275.857,Z 692.631,A -85,B 0,C 180,E1 11132.359,E2 11132.359} C_VEL
LIN {X 0,Y 278.458,Z 698.862,A -85,B 0,C 180,E1 11129.105,E2 11129.105} C_VEL
LIN {X 0,Y 280.631,Z 704.249,A -85,B 0,C 180,E1 11126.723,E2 11126.723} C_VEL
LIN {X 0,Y 288.949,Z 716.829,A -85,B 0,C 180,E1 11123.475,E2 11123.475} C_VEL
LIN {X 0,Y 296.441,Z 729.442,A -85,B 0,C 180,E1 11120.897,E2 11120.897} C_VEL
LIN {X 0,Y 301.319,Z 738.944,A -85,B 0,C 180,E1 11119.328,E2 11119.328} C_VEL
LIN {X 0,Y 302.411,Z 759.77,A -85,B 0,C 180,E1 11118.283,E2 11118.283} C_VEL
LIN {X 0,Y 293.997,Z 901.991,A -85,B 0,C 180,E1 11114.893,E2 11114.893} C_VEL
LIN {X 0,Y 291.651,Z 920.806,A -85,B 0,C 180,E1 11114.17,E2 11114.17} C_VEL
LIN {X 0,Y 288.404,Z 938.326,A -85,B 0,C 180,E1 11113.212,E2 11113.212} C_VEL
LIN {X 0,Y 284.329,Z 955.616,A -85,B 0,C 180,E1 11111.924,E2 11111.924} C_VEL
LIN {X 0,Y 279.516,Z 972.892,A -85,B 0,C 180,E1 11110.215,E2 11110.215} C_VEL
LIN {X 0,Y 274.39,Z 989.083,A -85,B 0,C 180,E1 11108.144,E2 11108.144} C_VEL
LIN {X 0,Y 269.334,Z 1003.698,A -85,B 0,C 180,E1 11105.781,E2 11105.781} C_VEL
LIN {X 0,Y 264.319,Z 1017.437,A -85,B 0,C 180,E1 11103.005,E2 11103.005} C_VEL
LIN {X 0,Y 259.588,Z 1030.175,A -85,B 0,C 180,E1 11099.793,E2 11099.793} C_VEL
LIN {X 0,Y 255.544,Z 1041.426,A -85,B 0,C 180,E1 11096.239,E2 11096.239} C_VEL
LIN {X 0,Y 252.351,Z 1051.199,A -85,B 0,C 180,E1 11092.356,E2 11092.356} C_VEL
LIN {X 0,Y 250.197,Z 1059.458,A -85,B 0,C 180,E1 11088.162,E2 11088.162} C_VEL
LIN {X 0,Y 249.178,Z 1065.805,A -85,B 0,C 180,E1 11083.931,E2 11083.931} C_VEL
LIN {X 0,Y 249.123,Z 1070.362,A -85,B 0,C 180,E1 11079.704,E2 11079.704} C_VEL
LIN {X 0,Y 249.62,Z 1073.076,A -85,B 0,C 180,E1 11075.747,E2 11075.747} C_VEL
LIN {X 0,Y 250.178,Z 1074.166,A -85,B 0,C 180,E1 11072.061,E2 11072.061} C_VEL
LIN {X 0,Y 250.322,Z 1073.858,A -85,B 0,C 180,E1 11068.855,E2 11068.855} C_VEL
LIN {X 0,Y 249.992,Z 1072.28,A -85,B 0,C 180,E1 11065.411,E2 11065.411} C_VEL
LIN {X 0,Y 249.458,Z 1068.635,A -85,B 0,C 180,E1 11061.239,E2 11061.239} C_VEL
LIN {X 0,Y 249.334,Z 1063.712,A -85,B 0,C 180,E1 11057.493,E2 11057.493} C_VEL
LIN {X 0,Y 250.023,Z 1055.59,A -85,B 0,C 180,E1 11053.026,E2 11053.026} C_VEL
LIN {X 0,Y 251.569,Z 1046.215,A -85,B 0,C 180,E1 11049.04,E2 11049.04} C_VEL
LIN {X 0,Y 253.963,Z 1035.271,A -85,B 0,C 180,E1 11045.334,E2 11045.334} C_VEL
LIN {X 0,Y 257.062,Z 1022.716,A -85,B 0,C 180,E1 11041.924,E2 11041.924} C_VEL
LIN {X 0,Y 260.573,Z 1009.14,A -85,B 0,C 180,E1 11038.945,E2 11038.945} C_VEL
LIN {X 0,Y 264.38,Z 994.238,A -85,B 0,C 180,E1 11036.306,E2 11036.306} C_VEL
LIN {X 0,Y 268.217,Z 978.211,A -85,B 0,C 180,E1 11034.046,E2 11034.046} C_VEL
LIN {X 0,Y 271.774,Z 961.866,A -85,B 0,C 180,E1 11032.225,E2 11032.225} C_VEL
LIN {X 0,Y 274.99,Z 944.809,A -85,B 0,C 180,E1 11030.752,E2 11030.752} C_VEL
LIN {X 0,Y 277.804,Z 926.501,A -85,B 0,C 180,E1 11029.586,E2 11029.586} C_VEL
LIN {X 0,Y 279.809,Z 907.373,A -85,B 0,C 180,E1 11028.737,E2 11028.737} C_VEL
LIN {X 0,Y 281.16,Z 880.236,A -85,B 0,C 180,E1 11028.002,E2 11028.002} C_VEL
LIN {X 0,Y 285.174,Z 791.387,A -85,B 0,C 180,E1 11025.834,E2 11025.834} C_VEL
LIN {X 0,Y 286.634,Z 780.007,A -85,B 0,C 180,E1 11025.354,E2 11025.354} C_VEL
LIN {X 0,Y 292.184,Z 756.705,A -85,B 0,C 180,E1 11024.058,E2 11024.058} C_VEL
LIN {X 0,Y 297.531,Z 730.584,A -85,B 0,C 180,E1 11021.711,E2 11021.711} C_VEL
LIN {X 0,Y 297.839,Z 717.253,A -85,B 0,C 180,E1 11017.782,E2 11017.782} C_VEL
LIN {X 0,Y 299.268,Z 709.917,A -85,B 0,C 180,E1 11015.059,E2 11015.059} C_VEL
LIN {X 0,Y 299.572,Z 708.876,A -85,B 0,C 180,E1 11014.569,E2 11014.569} C_VEL
LIN {X 0,Y 299.136,Z 710.685,A -85,B 0,C 180,E1 11010.98,E2 11010.98} C_VEL
LIN {X 0,Y 299.328,Z 714.178,A -85,B 0,C 180,E1 11008.315,E2 11008.315} C_VEL
LIN {X 0,Y 299.879,Z 718.769,A -85,B 0,C 180,E1 11005.809,E2 11005.809} C_VEL
LIN {X 0,Y 300.535,Z 724.98,A -85,B 0,C 180,E1 11003.322,E2 11003.322} C_VEL
LIN {X 0,Y 300.998,Z 732.429,A -85,B 0,C 180,E1 11001.022,E2 11001.022} C_VEL
LIN {X 0,Y 300.992,Z 734.478,A -85,B 0,C 180,E1 11000.505,E2 11000.505} C_VEL
LIN {X 0,Y 297.798,Z 751.472,A -85,B 0,C 180,E1 10997.941,E2 10997.941} C_VEL
LIN {X 0,Y 298.152,Z 756.234,A -85,B 0,C 180,E1 10997.478,E2 10997.478} C_VEL
LIN {X 0,Y 286.633,Z 863.562,A -85,B 0,C 180,E1 10993.721,E2 10993.721} C_VEL
LIN {X 0,Y 284.593,Z 892.141,A -85,B 0,C 180,E1 10992.446,E2 10992.446} C_VEL
LIN {X 0,Y 282.711,Z 908.747,A -85,B 0,C 180,E1 10991.319,E2 10991.319} C_VEL
LIN {X 0,Y 280.306,Z 923.566,A -85,B 0,C 180,E1 10989.962,E2 10989.962} C_VEL
LIN {X 0,Y 277.166,Z 938.34,A -85,B 0,C 180,E1 10988.192,E2 10988.192} C_VEL
LIN {X 0,Y 273.609,Z 951.928,A -85,B 0,C 180,E1 10986.083,E2 10986.083} C_VEL
LIN {X 0,Y 270.037,Z 963.336,A -85,B 0,C 180,E1 10983.821,E2 10983.821} C_VEL
LIN {X 0,Y 266.158,Z 974.191,A -85,B 0,C 180,E1 10981.076,E2 10981.076} C_VEL
LIN {X 0,Y 262.663,Z 982.71,A -85,B 0,C 180,E1 10978.254,E2 10978.254} C_VEL
LIN {X 0,Y 259.419,Z 989.844,A -85,B 0,C 180,E1 10975.135,E2 10975.135} C_VEL
LIN {X 0,Y 256.601,Z 995.275,A -85,B 0,C 180,E1 10971.784,E2 10971.784} C_VEL
LIN {X 0,Y 254.32,Z 998.988,A -85,B 0,C 180,E1 10968.224,E2 10968.224} C_VEL
LIN {X 0,Y 252.669,Z 1000.772,A -85,B 0,C 180,E1 10964.625,E2 10964.625} C_VEL
LIN {X 0,Y 251.623,Z 1000.782,A -85,B 0,C 180,E1 10960.983,E2 10960.983} C_VEL
LIN {X 0,Y 251.09,Z 998.883,A -85,B 0,C 180,E1 10957.277,E2 10957.277} C_VEL
LIN {X 0,Y 251.036,Z 995.384,A -85,B 0,C 180,E1 10953.761,E2 10953.761} C_VEL
LIN {X 0,Y 251.452,Z 989.742,A -85,B 0,C 180,E1 10950.095,E2 10950.095} C_VEL
LIN {X 0,Y 252.291,Z 982.645,A -85,B 0,C 180,E1 10946.744,E2 10946.744} C_VEL
LIN {X 0,Y 253.572,Z 973.545,A -85,B 0,C 180,E1 10943.458,E2 10943.458} C_VEL
LIN {X 0,Y 255.132,Z 963.212,A -85,B 0,C 180,E1 10940.539,E2 10940.539} C_VEL
LIN {X 0,Y 256.986,Z 951.013,A -85,B 0,C 180,E1 10937.787,E2 10937.787} C_VEL
LIN {X 0,Y 259.015,Z 936.755,A -85,B 0,C 180,E1 10935.259,E2 10935.259} C_VEL
LIN {X 0,Y 260.808,Z 922.295,A -85,B 0,C 180,E1 10933.247,E2 10933.247} C_VEL
LIN {X 0,Y 262.404,Z 907.103,A -85,B 0,C 180,E1 10931.591,E2 10931.591} C_VEL
LIN {X 0,Y 263.742,Z 889.933,A -85,B 0,C 180,E1 10930.209,E2 10930.209} C_VEL
LIN {X 0,Y 264.56,Z 873.049,A -85,B 0,C 180,E1 10929.272,E2 10929.272} C_VEL
LIN {X 0,Y 266.405,Z 822.098,A -85,B 0,C 180,E1 10927.501,E2 10927.501} C_VEL
LIN {X 0,Y 270.751,Z 738.453,A -85,B 0,C 180,E1 10924.749,E2 10924.749} C_VEL
LIN {X 0,Y 269.706,Z 729.368,A -85,B 0,C 180,E1 10924.237,E2 10924.237} C_VEL
LIN {X 0,Y 271.61,Z 705.697,A -85,B 0,C 180,E1 10920.777,E2 10920.777} C_VEL
LIN {X 0,Y 266.886,Z 687.863,A -85,B 0,C 180,E1 10917.319,E2 10917.319} C_VEL
LIN {X 0,Y 266.499,Z 686.536,A -85,B 0,C 180,E1 10916.999,E2 10916.999} C_VEL
LIN {X 0,Y 266.231,Z 686.751,A -85,B 0,C 180,E1 10916.64,E2 10916.64} C_VEL
LIN {X 0,Y 269.082,Z 697.827,A -85,B 0,C 180,E1 10913.236,E2 10913.236} C_VEL
LIN {X 0,Y 277.555,Z 715.098,A -85,B 0,C 180,E1 10911.249,E2 10911.249} C_VEL
LIN {X 0,Y 282.413,Z 746.301,A -85,B 0,C 180,E1 10909.534,E2 10909.534} C_VEL
LIN {X 0,Y 277.425,Z 857.925,A -85,B 0,C 180,E1 10906.718,E2 10906.718} C_VEL
LIN {X 0,Y 276.246,Z 875.3,A -85,B 0,C 180,E1 10905.934,E2 10905.934} C_VEL
LIN {X 0,Y 274.369,Z 892.386,A -85,B 0,C 180,E1 10904.78,E2 10904.78} C_VEL
LIN {X 0,Y 271.947,Z 908.661,A -85,B 0,C 180,E1 10903.285,E2 10903.285} C_VEL
LIN {X 0,Y 269.128,Z 923.756,A -85,B 0,C 180,E1 10901.465,E2 10901.465} C_VEL
LIN {X 0,Y 265.918,Z 938.446,A -85,B 0,C 180,E1 10899.196,E2 10899.196} C_VEL
LIN {X 0,Y 262.731,Z 951.516,A -85,B 0,C 180,E1 10896.646,E2 10896.646} C_VEL
LIN {X 0,Y 259.612,Z 963.182,A -85,B 0,C 180,E1 10893.755,E2 10893.755} C_VEL
LIN {X 0,Y 256.876,Z 973.073,A -85,B 0,C 180,E1 10890.67,E2 10890.67} C_VEL
LIN {X 0,Y 254.563,Z 981.564,A -85,B 0,C 180,E1 10887.299,E2 10887.299} C_VEL
LIN {X 0,Y 252.765,Z 988.513,A -85,B 0,C 180,E1 10883.642,E2 10883.642} C_VEL
LIN {X 0,Y 251.579,Z 993.899,A -85,B 0,C 180,E1 10879.698,E2 10879.698} C_VEL
LIN {X 0,Y 251.053,Z 997.439,A -85,B 0,C 180,E1 10875.705,E2 10875.705} C_VEL
LIN {X 0,Y 251.143,Z 999.126,A -85,B 0,C 180,E1 10871.669,E2 10871.669} C_VEL
LIN {X 0,Y 251.896,Z 999.075,A -85,B 0,C 180,E1 10867.601,E2 10867.601} C_VEL
LIN {X 0,Y 253.415,Z 997.223,A -85,B 0,C 180,E1 10863.523,E2 10863.523} C_VEL
LIN {X 0,Y 255.636,Z 993.629,A -85,B 0,C 180,E1 10859.699,E2 10859.699} C_VEL
LIN {X 0,Y 258.732,Z 988.154,A -85,B 0,C 180,E1 10855.921,E2 10855.921} C_VEL
LIN {X 0,Y 262.53,Z 980.99,A -85,B 0,C 180,E1 10852.39,E2 10852.39} C_VEL
LIN {X 0,Y 264.608,Z 976.8,A -85,B 0,C 180,E1 10850.749,E2 10850.749} C_VEL
LIN {X 0,Y 265.601,Z 973.084,A -85,B 0,C 180,E1 10849.298,E2 10849.298} C_VEL
LIN {X 0,Y 265.418,Z 963.859,A -85,B 0,C 180,E1 10845.705,E2 10845.705} C_VEL
LIN {X 0,Y 266.488,Z 959.278,A -85,B 0,C 180,E1 10844.379,E2 10844.379} C_VEL
LIN {X 0,Y 266.777,Z 958.552,A -85,B 0,C 180,E1 10844.208,E2 10844.208} C_VEL
LIN {X 0,Y 271.74,Z 946.17,A -85,B 0,C 180,E1 10841.675,E2 10841.675} C_VEL
LIN {X 0,Y 276.327,Z 933.014,A -85,B 0,C 180,E1 10839.557,E2 10839.557} C_VEL
LIN {X 0,Y 280.6,Z 918.384,A -85,B 0,C 180,E1 10837.717,E2 10837.717} C_VEL
LIN {X 0,Y 284.408,Z 902.376,A -85,B 0,C 180,E1 10836.164,E2 10836.164} C_VEL
LIN {X 0,Y 287.36,Z 886.09,A -85,B 0,C 180,E1 10834.975,E2 10834.975} C_VEL
LIN {X 0,Y 289.429,Z 868.986,A -85,B 0,C 180,E1 10834.094,E2 10834.094} C_VEL
LIN {X 0,Y 290.832,Z 847.559,A -85,B 0,C 180,E1 10833.409,E2 10833.409} C_VEL
LIN {X 0,Y 296.693,Z 753.739,A -85,B 0,C 180,E1 10831.123,E2 10831.123} C_VEL
LIN {X 0,Y 294.822,Z 742.162,A -85,B 0,C 180,E1 10830.184,E2 10830.184} C_VEL
LIN {X 0,Y 287.548,Z 728.417,A -85,B 0,C 180,E1 10827.603,E2 10827.603} C_VEL
LIN {X 0,Y 280.629,Z 717.11,A -85,B 0,C 180,E1 10824.918,E2 10824.918} C_VEL
LIN {X 0,Y 275.317,Z 709.19,A -85,B 0,C 180,E1 10822.642,E2 10822.642} C_VEL
LIN {X 0,Y 271.418,Z 703.574,A -85,B 0,C 180,E1 10820.768,E2 10820.768} C_VEL
LIN {X 0,Y 268.7,Z 699.371,A -85,B 0,C 180,E1 10819.228,E2 10819.228} C_VEL
LIN {X 0,Y 266.798,Z 693.545,A -85,B 0,C 180,E1 10815.432,E2 10815.432} C_VEL
LIN {X 0,Y 265.404,Z 689.755,A -85,B 0,C 180,E1 10812.401,E2 10812.401} C_VEL
LIN {X 0,Y 264.329,Z 686.685,A -85,B 0,C 180,E1 10809.581,E2 10809.581} C_VEL
LIN {X 0,Y 263.224,Z 683.339,A -85,B 0,C 180,E1 10805.45,E2 10805.45} C_VEL
LIN {X 0,Y 262.125,Z 680.058,A -85,B 0,C 180,E1 10798.252,E2 10798.252} C_VEL
LIN {X 0,Y 262.178,Z 679.899,A -85,B 0,C 180,E1 10793.211,E2 10793.211} C_VEL
LIN {X 0,Y 262.651,Z 680.941,A -85,B 0,C 180,E1 10789.694,E2 10789.694} C_VEL
LIN {X 0,Y 264.747,Z 685.133,A -85,B 0,C 180,E1 10782.868,E2 10782.868} C_VEL
LIN {X 0,Y 266.698,Z 689.504,A -85,B 0,C 180,E1 10778.675,E2 10778.675} C_VEL
LIN {X 0,Y 268.552,Z 694.03,A -85,B 0,C 180,E1 10775.291,E2 10775.291} C_VEL
LIN {X 0,Y 270.483,Z 698.573,A -85,B 0,C 180,E1 10772.48,E2 10772.48} C_VEL
LIN {X 0,Y 272.917,Z 704.206,A -85,B 0,C 180,E1 10769.57,E2 10769.57} C_VEL
LIN {X 0,Y 279.183,Z 713.425,A -85,B 0,C 180,E1 10766.713,E2 10766.713} C_VEL
LIN {X 0,Y 285.936,Z 723.716,A -85,B 0,C 180,E1 10764.054,E2 10764.054} C_VEL
LIN {X 0,Y 292.942,Z 735.958,A -85,B 0,C 180,E1 10761.534,E2 10761.534} C_VEL
LIN {X 0,Y 296.44,Z 742.993,A -85,B 0,C 180,E1 10760.349,E2 10760.349} C_VEL
LIN {X 0,Y 297.251,Z 760.957,A -85,B 0,C 180,E1 10759.439,E2 10759.439} C_VEL
LIN {X 0,Y 288.558,Z 901.285,A -85,B 0,C 180,E1 10756.06,E2 10756.06} C_VEL
LIN {X 0,Y 286.13,Z 920.022,A -85,B 0,C 180,E1 10755.334,E2 10755.334} C_VEL
LIN {X 0,Y 282.612,Z 938.238,A -85,B 0,C 180,E1 10754.325,E2 10754.325} C_VEL
LIN {X 0,Y 278.121,Z 956.355,A -85,B 0,C 180,E1 10752.942,E2 10752.942} C_VEL
LIN {X 0,Y 273.143,Z 973.305,A -85,B 0,C 180,E1 10751.216,E2 10751.216} C_VEL
LIN {X 0,Y 267.822,Z 989.245,A -85,B 0,C 180,E1 10749.118,E2 10749.118} C_VEL
LIN {X 0,Y 262.35,Z 1004.199,A -85,B 0,C 180,E1 10746.615,E2 10746.615} C_VEL
LIN {X 0,Y 257.131,Z 1017.642,A -85,B 0,C 180,E1 10743.783,E2 10743.783} C_VEL
LIN {X 0,Y 252.191,Z 1030.11,A -85,B 0,C 180,E1 10740.496,E2 10740.496} C_VEL
LIN {X 0,Y 247.951,Z 1041.14,A -85,B 0,C 180,E1 10736.848,E2 10736.848} C_VEL
LIN {X 0,Y 244.59,Z 1050.726,A -85,B 0,C 180,E1 10732.851,E2 10732.851} C_VEL
LIN {X 0,Y 242.308,Z 1058.82,A -85,B 0,C 180,E1 10728.525,E2 10728.525} C_VEL
LIN {X 0,Y 241.192,Z 1065.31,A -85,B 0,C 180,E1 10723.912,E2 10723.912} C_VEL
LIN {X 0,Y 241.19,Z 1069.758,A -85,B 0,C 180,E1 10719.379,E2 10719.379} C_VEL
LIN {X 0,Y 241.776,Z 1072.195,A -85,B 0,C 180,E1 10715.219,E2 10715.219} C_VEL
LIN {X 0,Y 242.312,Z 1072.985,A -85,B 0,C 180,E1 10711.655,E2 10711.655} C_VEL
LIN {X 0,Y 242.403,Z 1072.551,A -85,B 0,C 180,E1 10708.581,E2 10708.581} C_VEL
LIN {X 0,Y 242.013,Z 1070.796,A -85,B 0,C 180,E1 10705.022,E2 10705.022} C_VEL
LIN {X 0,Y 241.438,Z 1067.335,A -85,B 0,C 180,E1 10700.705,E2 10700.705} C_VEL
LIN {X 0,Y 241.375,Z 1062.471,A -85,B 0,C 180,E1 10696.83,E2 10696.83} C_VEL
LIN {X 0,Y 242.03,Z 1055.639,A -85,B 0,C 180,E1 10692.943,E2 10692.943} C_VEL
LIN {X 0,Y 243.379,Z 1047.377,A -85,B 0,C 180,E1 10689.309,E2 10689.309} C_VEL
LIN {X 0,Y 246.283,Z 1034.169,A -85,B 0,C 180,E1 10684.768,E2 10684.768} C_VEL
LIN {X 0,Y 249.54,Z 1021.589,A -85,B 0,C 180,E1 10681.26,E2 10681.26} C_VEL
LIN {X 0,Y 253.198,Z 1008.059,A -85,B 0,C 180,E1 10678.216,E2 10678.216} C_VEL
LIN {X 0,Y 257.177,Z 993.08,A -85,B 0,C 180,E1 10675.509,E2 10675.509} C_VEL
LIN {X 0,Y 261.182,Z 976.964,A -85,B 0,C 180,E1 10673.193,E2 10673.193} C_VEL
LIN {X 0,Y 264.875,Z 960.49,A -85,B 0,C 180,E1 10671.337,E2 10671.337} C_VEL
LIN {X 0,Y 268.319,Z 942.653,A -85,B 0,C 180,E1 10669.789,E2 10669.789} C_VEL
LIN {X 0,Y 271.227,Z 923.955,A -85,B 0,C 180,E1 10668.612,E2 10668.612} C_VEL
LIN {X 0,Y 273.183,Z 904.927,A -85,B 0,C 180,E1 10667.781,E2 10667.781} C_VEL
LIN {X 0,Y 274.877,Z 869.393,A -85,B 0,C 180,E1 10666.848,E2 10666.848} C_VEL
LIN {X 0,Y 276.708,Z 831.712,A -85,B 0,C 180,E1 10665.881,E2 10665.881} C_VEL
LIN {X 0,Y 283.274,Z 779.789,A -85,B 0,C 180,E1 10663.868,E2 10663.868} C_VEL
LIN {X 0,Y 288.799,Z 758.139,A -85,B 0,C 180,E1 10662.632,E2 10662.632} C_VEL
LIN {X 0,Y 294.025,Z 735.062,A -85,B 0,C 180,E1 10660.505,E2 10660.505} C_VEL
LIN {X 0,Y 294.853,Z 723.174,A -85,B 0,C 180,E1 10656.885,E2 10656.885} C_VEL
LIN {X 0,Y 296.431,Z 716.419,A -85,B 0,C 180,E1 10654.342,E2 10654.342} C_VEL
LIN {X 0,Y 295.926,Z 718.069,A -85,B 0,C 180,E1 10651.127,E2 10651.127} C_VEL
LIN {X 0,Y 295.858,Z 721.408,A -85,B 0,C 180,E1 10648.516,E2 10648.516} C_VEL
LIN {X 0,Y 296.152,Z 725.946,A -85,B 0,C 180,E1 10646.033,E2 10646.033} C_VEL
LIN {X 0,Y 296.493,Z 731.873,A -85,B 0,C 180,E1 10643.659,E2 10643.659} C_VEL
LIN {X 0,Y 296.638,Z 738.927,A -85,B 0,C 180,E1 10641.487,E2 10641.487} C_VEL
LIN {X 0,Y 293.731,Z 753.262,A -85,B 0,C 180,E1 10639.306,E2 10639.306} C_VEL
LIN {X 0,Y 294.005,Z 758.451,A -85,B 0,C 180,E1 10638.765,E2 10638.765} C_VEL
LIN {X 0,Y 281.865,Z 864.312,A -85,B 0,C 180,E1 10635.008,E2 10635.008} C_VEL
LIN {X 0,Y 279.523,Z 893.589,A -85,B 0,C 180,E1 10633.668,E2 10633.668} C_VEL
LIN {X 0,Y 277.421,Z 910.62,A -85,B 0,C 180,E1 10632.488,E2 10632.488} C_VEL
LIN {X 0,Y 274.836,Z 925.239,A -85,B 0,C 180,E1 10631.117,E2 10631.117} C_VEL
LIN {X 0,Y 271.481,Z 939.907,A -85,B 0,C 180,E1 10629.326,E2 10629.326} C_VEL
LIN {X 0,Y 267.661,Z 953.376,A -85,B 0,C 180,E1 10627.188,E2 10627.188} C_VEL
LIN {X 0,Y 263.682,Z 965.241,A -85,B 0,C 180,E1 10624.785,E2 10624.785} C_VEL
LIN {X 0,Y 259.832,Z 975.209,A -85,B 0,C 180,E1 10622.205,E2 10622.205} C_VEL
LIN {X 0,Y 255.988,Z 983.937,A -85,B 0,C 180,E1 10619.273,E2 10619.273} C_VEL
LIN {X 0,Y 252.523,Z 990.992,A -85,B 0,C 180,E1 10616.14,E2 10616.14} C_VEL
LIN {X 0,Y 249.556,Z 996.263,A -85,B 0,C 180,E1 10612.865,E2 10612.865} C_VEL
LIN {X 0,Y 247.034,Z 1000.07,A -85,B 0,C 180,E1 10609.269,E2 10609.269} C_VEL
LIN {X 0,Y 245.154,Z 1002.03,A -85,B 0,C 180,E1 10605.594,E2 10605.594} C_VEL
LIN {X 0,Y 243.908,Z 1002.196,A -85,B 0,C 180,E1 10601.847,E2 10601.847} C_VEL
LIN {X 0,Y 243.261,Z 1000.686,A -85,B 0,C 180,E1 10598.268,E2 10598.268} C_VEL
LIN {X 0,Y 243.074,Z 997.197,A -85,B 0,C 180,E1 10594.411,E2 10594.411} C_VEL
LIN {X 0,Y 243.353,Z 992.449,A -85,B 0,C 180,E1 10590.998,E2 10590.998} C_VEL
LIN {X 0,Y 244.16,Z 985.233,A -85,B 0,C 180,E1 10587.278,E2 10587.278} C_VEL
LIN {X 0,Y 245.309,Z 976.989,A -85,B 0,C 180,E1 10584.06,E2 10584.06} C_VEL
LIN {X 0,Y 246.939,Z 966.436,A -85,B 0,C 180,E1 10580.828,E2 10580.828} C_VEL
LIN {X 0,Y 248.736,Z 954.904,A -85,B 0,C 180,E1 10578.045,E2 10578.045} C_VEL
LIN {X 0,Y 250.662,Z 942.119,A -85,B 0,C 180,E1 10575.563,E2 10575.563} C_VEL
LIN {X 0,Y 252.673,Z 927.113,A -85,B 0,C 180,E1 10573.271,E2 10573.271} C_VEL
LIN {X 0,Y 254.36,Z 912.32,A -85,B 0,C 180,E1 10571.51,E2 10571.51} C_VEL
LIN {X 0,Y 255.84,Z 895.694,A -85,B 0,C 180,E1 10570.003,E2 10570.003} C_VEL
LIN {X 0,Y 256.916,Z 877.346,A -85,B 0,C 180,E1 10568.849,E2 10568.849} C_VEL
LIN {X 0,Y 258.251,Z 837.356,A -85,B 0,C 180,E1 10567.348,E2 10567.348} C_VEL
LIN {X 0,Y 263.543,Z 739.399,A -85,B 0,C 180,E1 10564.013,E2 10564.013} C_VEL
LIN {X 0,Y 262.549,Z 730.383,A -85,B 0,C 180,E1 10563.486,E2 10563.486} C_VEL
LIN {X 0,Y 264.372,Z 708.116,A -85,B 0,C 180,E1 10560.2,E2 10560.2} C_VEL
LIN {X 0,Y 260.143,Z 691.812,A -85,B 0,C 180,E1 10556.94,E2 10556.94} C_VEL
LIN {X 0,Y 259.784,Z 692.008,A -85,B 0,C 180,E1 10556.518,E2 10556.518} C_VEL
LIN {X 0,Y 261.239,Z 697.848,A -85,B 0,C 180,E1 10554.658,E2 10554.658} C_VEL
LIN {X 0,Y 270.714,Z 716.767,A -85,B 0,C 180,E1 10552.3,E2 10552.3} C_VEL
LIN {X 0,Y 271.688,Z 719.66,A -85,B 0,C 180,E1 10552.044,E2 10552.044} C_VEL
LIN {X 0,Y 275.897,Z 747.556,A -85,B 0,C 180,E1 10550.474,E2 10550.474} C_VEL
LIN {X 0,Y 270.732,Z 858.415,A -85,B 0,C 180,E1 10547.629,E2 10547.629} C_VEL
LIN {X 0,Y 269.515,Z 875.785,A -85,B 0,C 180,E1 10546.836,E2 10546.836} C_VEL
LIN {X 0,Y 267.651,Z 892.264,A -85,B 0,C 180,E1 10545.715,E2 10545.715} C_VEL
LIN {X 0,Y 265.122,Z 908.748,A -85,B 0,C 180,E1 10544.19,E2 10544.19} C_VEL
LIN {X 0,Y 262.185,Z 924.057,A -85,B 0,C 180,E1 10542.332,E2 10542.332} C_VEL
LIN {X 0,Y 259.033,Z 937.993,A -85,B 0,C 180,E1 10540.165,E2 10540.165} C_VEL
LIN {X 0,Y 255.632,Z 951.441,A -85,B 0,C 180,E1 10537.53,E2 10537.53} C_VEL
LIN {X 0,Y 252.555,Z 962.658,A -85,B 0,C 180,E1 10534.77,E2 10534.77} C_VEL
LIN {X 0,Y 249.608,Z 972.833,A -85,B 0,C 180,E1 10531.607,E2 10531.607} C_VEL
LIN {X 0,Y 247.09,Z 981.579,A -85,B 0,C 180,E1 10528.145,E2 10528.145} C_VEL
LIN {X 0,Y 245.122,Z 988.858,A -85,B 0,C 180,E1 10524.383,E2 10524.383} C_VEL
LIN {X 0,Y 243.849,Z 994.21,A -85,B 0,C 180,E1 10520.561,E2 10520.561} C_VEL
LIN {X 0,Y 243.178,Z 998.059,A -85,B 0,C 180,E1 10516.447,E2 10516.447} C_VEL
LIN {X 0,Y 243.175,Z 1000.151,A -85,B 0,C 180,E1 10512.287,E2 10512.287} C_VEL
LIN {X 0,Y 243.852,Z 1000.447,A -85,B 0,C 180,E1 10508.092,E2 10508.092} C_VEL
LIN {X 0,Y 245.317,Z 998.927,A -85,B 0,C 180,E1 10503.885,E2 10503.885} C_VEL
LIN {X 0,Y 247.637,Z 995.612,A -85,B 0,C 180,E1 10499.775,E2 10499.775} C_VEL
LIN {X 0,Y 250.624,Z 990.757,A -85,B 0,C 180,E1 10496.047,E2 10496.047} C_VEL
LIN {X 0,Y 254.376,Z 984.14,A -85,B 0,C 180,E1 10492.465,E2 10492.465} C_VEL
LIN {X 0,Y 258.622,Z 976.091,A -85,B 0,C 180,E1 10489.204,E2 10489.204} C_VEL
LIN {X 0,Y 263.327,Z 966.393,A -85,B 0,C 180,E1 10486.174,E2 10486.174} C_VEL
LIN {X 0,Y 266.777,Z 958.552,A -85,B 0,C 180,E1 10484.208,E2 10484.208} C_VEL
LIN {X 0,Y 268.11,Z 953.607,A -85,B 0,C 180,E1 10482.962,E2 10482.962} C_VEL
LIN {X 0,Y 268.621,Z 941.653,A -85,B 0,C 180,E1 10479.819,E2 10479.819} C_VEL
LIN {X 0,Y 269.799,Z 935.934,A -85,B 0,C 180,E1 10478.722,E2 10478.722} C_VEL
LIN {X 0,Y 270.091,Z 935.064,A -85,B 0,C 180,E1 10478.586,E2 10478.586} C_VEL
LIN {X 0,Y 274.499,Z 920.914,A -85,B 0,C 180,E1 10476.742,E2 10476.742} C_VEL
LIN {X 0,Y 278.374,Z 905.661,A -85,B 0,C 180,E1 10475.202,E2 10475.202} C_VEL
LIN {X 0,Y 281.654,Z 888.906,A -85,B 0,C 180,E1 10473.922,E2 10473.922} C_VEL
LIN {X 0,Y 283.987,Z 871.804,A -85,B 0,C 180,E1 10472.984,E2 10472.984} C_VEL
LIN {X 0,Y 285.376,Z 853.04,A -85,B 0,C 180,E1 10472.331,E2 10472.331} C_VEL
LIN {X 0,Y 291.715,Z 755.351,A -85,B 0,C 180,E1 10469.915,E2 10469.915} C_VEL
LIN {X 0,Y 290.36,Z 746.757,A -85,B 0,C 180,E1 10469.189,E2 10469.189} C_VEL
LIN {X 0,Y 283.818,Z 734.145,A -85,B 0,C 180,E1 10466.747,E2 10466.747} C_VEL
LIN {X 0,Y 277.421,Z 723.442,A -85,B 0,C 180,E1 10464.147,E2 10464.147} C_VEL
LIN {X 0,Y 272.508,Z 715.844,A -85,B 0,C 180,E1 10461.922,E2 10461.922} C_VEL
LIN {X 0,Y 268.721,Z 710.274,A -85,B 0,C 180,E1 10460.018,E2 10460.018} C_VEL
LIN {X 0,Y 265.547,Z 705.701,A -85,B 0,C 180,E1 10458.268,E2 10458.268} C_VEL
LIN {X 0,Y 261.575,Z 700.03,A -85,B 0,C 180,E1 10455.748,E2 10455.748} C_VEL
LIN {X 0,Y 259.901,Z 695.5,A -85,B 0,C 180,E1 10452.216,E2 10452.216} C_VEL
LIN {X 0,Y 258.922,Z 692.508,A -85,B 0,C 180,E1 10449.334,E2 10449.334} C_VEL
LIN {X 0,Y 257.94,Z 689.329,A -85,B 0,C 180,E1 10445.338,E2 10445.338} C_VEL
LIN {X 0,Y 256.966,Z 686.174,A -85,B 0,C 180,E1 10438.217,E2 10438.217} C_VEL
LIN {X 0,Y 257.108,Z 686.091,A -85,B 0,C 180,E1 10433.076,E2 10433.076} C_VEL
LIN {X 0,Y 257.544,Z 687.113,A -85,B 0,C 180,E1 10429.713,E2 10429.713} C_VEL
LIN {X 0,Y 259.56,Z 691.234,A -85,B 0,C 180,E1 10422.977,E2 10422.977} C_VEL
LIN {X 0,Y 261.466,Z 695.683,A -85,B 0,C 180,E1 10418.698,E2 10418.698} C_VEL
LIN {X 0,Y 263.289,Z 700.179,A -85,B 0,C 180,E1 10415.309,E2 10415.309} C_VEL
LIN {X 0,Y 264.918,Z 703.764,A -85,B 0,C 180,E1 10413.131,E2 10413.131} C_VEL
LIN {X 0,Y 270.792,Z 711.935,A -85,B 0,C 180,E1 10409.98,E2 10409.98} C_VEL
LIN {X 0,Y 276.113,Z 719.842,A -85,B 0,C 180,E1 10407.47,E2 10407.47} C_VEL
LIN {X 0,Y 282.603,Z 730.036,A -85,B 0,C 180,E1 10404.782,E2 10404.782} C_VEL
LIN {X 0,Y 289.384,Z 742.224,A -85,B 0,C 180,E1 10402.236,E2 10402.236} C_VEL
LIN {X 0,Y 291.672,Z 747.087,A -85,B 0,C 180,E1 10401.406,E2 10401.406} C_VEL
LIN {X 0,Y 292.218,Z 762.158,A -85,B 0,C 180,E1 10400.635,E2 10400.635} C_VEL
LIN {X 0,Y 283.284,Z 900.465,A -85,B 0,C 180,E1 10397.281,E2 10397.281} C_VEL
LIN {X 0,Y 280.777,Z 919.187,A -85,B 0,C 180,E1 10396.552,E2 10396.552} C_VEL
LIN {X 0,Y 277.23,Z 936.958,A -85,B 0,C 180,E1 10395.569,E2 10395.569} C_VEL
LIN {X 0,Y 272.572,Z 955.122,A -85,B 0,C 180,E1 10394.183,E2 10394.183} C_VEL
LIN {X 0,Y 267.647,Z 971.273,A -85,B 0,C 180,E1 10392.544,E2 10392.544} C_VEL
LIN {X 0,Y 262.056,Z 987.375,A -85,B 0,C 180,E1 10390.437,E2 10390.437} C_VEL
LIN {X 0,Y 256.508,Z 1001.893,A -85,B 0,C 180,E1 10388.015,E2 10388.015} C_VEL
LIN {X 0,Y 250.751,Z 1016.017,A -85,B 0,C 180,E1 10385.043,E2 10385.043} C_VEL
LIN {X 0,Y 245.468,Z 1028.56,A -85,B 0,C 180,E1 10381.698,E2 10381.698} C_VEL
LIN {X 0,Y 240.881,Z 1039.635,A -85,B 0,C 180,E1 10377.972,E2 10377.972} C_VEL
LIN {X 0,Y 237.16,Z 1049.387,A -85,B 0,C 180,E1 10373.814,E2 10373.814} C_VEL
LIN {X 0,Y 234.631,Z 1057.413,A -85,B 0,C 180,E1 10369.413,E2 10369.413} C_VEL
LIN {X 0,Y 233.301,Z 1063.943,A -85,B 0,C 180,E1 10364.646,E2 10364.646} C_VEL
LIN {X 0,Y 233.192,Z 1068.503,A -85,B 0,C 180,E1 10359.875,E2 10359.875} C_VEL
LIN {X 0,Y 233.763,Z 1070.931,A -85,B 0,C 180,E1 10355.645,E2 10355.645} C_VEL
LIN {X 0,Y 234.363,Z 1071.773,A -85,B 0,C 180,E1 10351.955,E2 10351.955} C_VEL
LIN {X 0,Y 234.506,Z 1071.371,A -85,B 0,C 180,E1 10348.778,E2 10348.778} C_VEL
LIN {X 0,Y 234.099,Z 1069.662,A -85,B 0,C 180,E1 10345.099,E2 10345.099} C_VEL
LIN {X 0,Y 233.46,Z 1066.516,A -85,B 0,C 180,E1 10340.633,E2 10340.633} C_VEL
LIN {X 0,Y 233.403,Z 1061.79,A -85,B 0,C 180,E1 10336.513,E2 10336.513} C_VEL
LIN {X 0,Y 234.108,Z 1055.456,A -85,B 0,C 180,E1 10332.604,E2 10332.604} C_VEL
LIN {X 0,Y 235.843,Z 1046.345,A -85,B 0,C 180,E1 10328.355,E2 10328.355} C_VEL
LIN {X 0,Y 238.293,Z 1036.13,A -85,B 0,C 180,E1 10324.66,E2 10324.66} C_VEL
LIN {X 0,Y 241.333,Z 1024.5,A -85,B 0,C 180,E1 10321.275,E2 10321.275} C_VEL
LIN {X 0,Y 244.739,Z 1011.899,A -85,B 0,C 180,E1 10318.311,E2 10318.311} C_VEL
LIN {X 0,Y 248.736,Z 996.871,A -85,B 0,C 180,E1 10315.473,E2 10315.473} C_VEL
LIN {X 0,Y 253.4,Z 978.881,A -85,B 0,C 180,E1 10312.722,E2 10312.722} C_VEL
LIN {X 0,Y 257.383,Z 962.19,A -85,B 0,C 180,E1 10310.712,E2 10310.712} C_VEL
LIN {X 0,Y 261.025,Z 944.437,A -85,B 0,C 180,E1 10309.078,E2 10309.078} C_VEL
LIN {X 0,Y 264.153,Z 925.645,A -85,B 0,C 180,E1 10307.815,E2 10307.815} C_VEL
LIN {X 0,Y 266.325,Z 906.257,A -85,B 0,C 180,E1 10306.917,E2 10306.917} C_VEL
LIN {X 0,Y 267.755,Z 880.07,A -85,B 0,C 180,E1 10306.174,E2 10306.174} C_VEL
LIN {X 0,Y 268.599,Z 868.633,A -85,B 0,C 180,E1 10305.791,E2 10305.791} C_VEL
LIN {X 0,Y 280.254,Z 781.379,A -85,B 0,C 180,E1 10302.394,E2 10302.394} C_VEL
LIN {X 0,Y 281.782,Z 774.156,A -85,B 0,C 180,E1 10302.055,E2 10302.055} C_VEL
LIN {X 0,Y 285.66,Z 759.819,A -85,B 0,C 180,E1 10301.188,E2 10301.188} C_VEL
LIN {X 0,Y 290.656,Z 739.874,A -85,B 0,C 180,E1 10299.362,E2 10299.362} C_VEL
LIN {X 0,Y 291.84,Z 729.434,A -85,B 0,C 180,E1 10296.106,E2 10296.106} C_VEL
LIN {X 0,Y 293.233,Z 723.979,A -85,B 0,C 180,E1 10294,E2 10294} C_VEL
LIN {X 0,Y 292.682,Z 725.425,A -85,B 0,C 180,E1 10291.282,E2 10291.282} C_VEL
LIN {X 0,Y 292.471,Z 728.513,A -85,B 0,C 180,E1 10288.818,E2 10288.818} C_VEL
LIN {X 0,Y 292.496,Z 732.895,A -85,B 0,C 180,E1 10286.384,E2 10286.384} C_VEL
LIN {X 0,Y 292.554,Z 739.489,A -85,B 0,C 180,E1 10283.783,E2 10283.783} C_VEL
LIN {X 0,Y 292.385,Z 744.075,A -85,B 0,C 180,E1 10282.413,E2 10282.413} C_VEL
LIN {X 0,Y 289.946,Z 755.142,A -85,B 0,C 180,E1 10280.712,E2 10280.712} C_VEL
LIN {X 0,Y 290.167,Z 760.72,A -85,B 0,C 180,E1 10280.103,E2 10280.103} C_VEL
LIN {X 0,Y 277.372,Z 865.264,A -85,B 0,C 180,E1 10276.35,E2 10276.35} C_VEL
LIN {X 0,Y 274.723,Z 894.944,A -85,B 0,C 180,E1 10274.962,E2 10274.962} C_VEL
LIN {X 0,Y 272.514,Z 911.581,A -85,B 0,C 180,E1 10273.797,E2 10273.797} C_VEL
LIN {X 0,Y 269.749,Z 926.243,A -85,B 0,C 180,E1 10272.414,E2 10272.414} C_VEL
LIN {X 0,Y 265.963,Z 941.654,A -85,B 0,C 180,E1 10270.505,E2 10270.505} C_VEL
LIN {X 0,Y 261.872,Z 954.994,A -85,B 0,C 180,E1 10268.342,E2 10268.342} C_VEL
LIN {X 0,Y 257.797,Z 966.33,A -85,B 0,C 180,E1 10266.011,E2 10266.011} C_VEL
LIN {X 0,Y 253.323,Z 977.07,A -85,B 0,C 180,E1 10263.167,E2 10263.167} C_VEL
LIN {X 0,Y 249.28,Z 985.555,A -85,B 0,C 180,E1 10260.229,E2 10260.229} C_VEL
LIN {X 0,Y 245.342,Z 992.864,A -85,B 0,C 180,E1 10256.836,E2 10256.836} C_VEL
LIN {X 0,Y 242.071,Z 998.134,A -85,B 0,C 180,E1 10253.358,E2 10253.358} C_VEL
LIN {X 0,Y 239.378,Z 1001.739,A -85,B 0,C 180,E1 10249.653,E2 10249.653} C_VEL
LIN {X 0,Y 237.304,Z 1003.515,A -85,B 0,C 180,E1 10245.719,E2 10245.719} C_VEL
LIN {X 0,Y 236.033,Z 1003.488,A -85,B 0,C 180,E1 10241.986,E2 10241.986} C_VEL
LIN {X 0,Y 235.306,Z 1001.59,A -85,B 0,C 180,E1 10238.041,E2 10238.041} C_VEL
LIN {X 0,Y 235.139,Z 998.11,A -85,B 0,C 180,E1 10234.295,E2 10234.295} C_VEL
LIN {X 0,Y 235.475,Z 992.671,A -85,B 0,C 180,E1 10230.491,E2 10230.491} C_VEL
LIN {X 0,Y 236.295,Z 985.684,A -85,B 0,C 180,E1 10226.912,E2 10226.912} C_VEL
LIN {X 0,Y 237.639,Z 976.398,A -85,B 0,C 180,E1 10223.311,E2 10223.311} C_VEL
LIN {X 0,Y 239.245,Z 966.34,A -85,B 0,C 180,E1 10220.251,E2 10220.251} C_VEL
LIN {X 0,Y 241.191,Z 954.294,A -85,B 0,C 180,E1 10217.326,E2 10217.326} C_VEL
LIN {X 0,Y 243.212,Z 941.09,A -85,B 0,C 180,E1 10214.787,E2 10214.787} C_VEL
LIN {X 0,Y 245.16,Z 926.885,A -85,B 0,C 180,E1 10212.612,E2 10212.612} C_VEL
LIN {X 0,Y 247.059,Z 910.33,A -85,B 0,C 180,E1 10210.661,E2 10210.661} C_VEL
LIN {X 0,Y 248.462,Z 894.176,A -85,B 0,C 180,E1 10209.245,E2 10209.245} C_VEL
LIN {X 0,Y 249.459,Z 877.054,A -85,B 0,C 180,E1 10208.182,E2 10208.182} C_VEL
LIN {X 0,Y 251.437,Z 826.464,A -85,B 0,C 180,E1 10206.272,E2 10206.272} C_VEL
LIN {X 0,Y 256.333,Z 740.277,A -85,B 0,C 180,E1 10203.25,E2 10203.25} C_VEL
LIN {X 0,Y 255.402,Z 731.301,A -85,B 0,C 180,E1 10202.701,E2 10202.701} C_VEL
LIN {X 0,Y 257.173,Z 710.553,A -85,B 0,C 180,E1 10199.589,E2 10199.589} C_VEL
LIN {X 0,Y 253.672,Z 697.048,A -85,B 0,C 180,E1 10196.828,E2 10196.828} C_VEL
LIN {X 0,Y 253.277,Z 697.294,A -85,B 0,C 180,E1 10196.395,E2 10196.395} C_VEL
LIN {X 0,Y 254.135,Z 699.465,A -85,B 0,C 180,E1 10195.946,E2 10195.946} C_VEL
LIN {X 0,Y 261.678,Z 713.963,A -85,B 0,C 180,E1 10193.972,E2 10193.972} C_VEL
LIN {X 0,Y 265.601,Z 722.53,A -85,B 0,C 180,E1 10192.976,E2 10192.976} C_VEL
LIN {X 0,Y 269.432,Z 748.745,A -85,B 0,C 180,E1 10191.452,E2 10191.452} C_VEL
LIN {X 0,Y 264.081,Z 859.031,A -85,B 0,C 180,E1 10188.574,E2 10188.574} C_VEL
LIN {X 0,Y 262.809,Z 876.497,A -85,B 0,C 180,E1 10187.763,E2 10187.763} C_VEL
LIN {X 0,Y 260.755,Z 893.797,A -85,B 0,C 180,E1 10186.555,E2 10186.555} C_VEL
LIN {X 0,Y 258.19,Z 909.764,A -85,B 0,C 180,E1 10185.039,E2 10185.039} C_VEL
LIN {X 0,Y 255.131,Z 925.055,A -85,B 0,C 180,E1 10183.139,E2 10183.139} C_VEL
LIN {X 0,Y 251.779,Z 939.259,A -85,B 0,C 180,E1 10180.874,E2 10180.874} C_VEL
LIN {X 0,Y 248.298,Z 952.449,A -85,B 0,C 180,E1 10178.219,E2 10178.219} C_VEL
LIN {X 0,Y 245.029,Z 963.858,A -85,B 0,C 180,E1 10175.333,E2 10175.333} C_VEL
LIN {X 0,Y 242.001,Z 973.872,A -85,B 0,C 180,E1 10172.132,E2 10172.132} C_VEL
LIN {X 0,Y 239.362,Z 982.637,A -85,B 0,C 180,E1 10168.564,E2 10168.564} C_VEL
LIN {X 0,Y 237.296,Z 989.937,A -85,B 0,C 180,E1 10164.682,E2 10164.682} C_VEL
LIN {X 0,Y 235.96,Z 995.321,A -85,B 0,C 180,E1 10160.734,E2 10160.734} C_VEL
LIN {X 0,Y 235.259,Z 999.199,A -85,B 0,C 180,E1 10156.483,E2 10156.483} C_VEL
LIN {X 0,Y 235.266,Z 1001.326,A -85,B 0,C 180,E1 10152.174,E2 10152.174} C_VEL
LIN {X 0,Y 235.997,Z 1001.676,A -85,B 0,C 180,E1 10147.848,E2 10147.848} C_VEL
LIN {X 0,Y 237.562,Z 1000.202,A -85,B 0,C 180,E1 10143.505,E2 10143.505} C_VEL
LIN {X 0,Y 239.906,Z 997.099,A -85,B 0,C 180,E1 10139.439,E2 10139.439} C_VEL
LIN {X 0,Y 243.191,Z 992.169,A -85,B 0,C 180,E1 10135.433,E2 10135.433} C_VEL
LIN {X 0,Y 247.232,Z 985.464,A -85,B 0,C 180,E1 10131.683,E2 10131.683} C_VEL
LIN {X 0,Y 251.942,Z 977.019,A -85,B 0,C 180,E1 10128.186,E2 10128.186} C_VEL
LIN {X 0,Y 256.912,Z 967.273,A -85,B 0,C 180,E1 10125.099,E2 10125.099} C_VEL
LIN {X 0,Y 261.908,Z 956.305,A -85,B 0,C 180,E1 10122.4,E2 10122.4} C_VEL
LIN {X 0,Y 266.819,Z 944.127,A -85,B 0,C 180,E1 10120.036,E2 10120.036} C_VEL
LIN {X 0,Y 270.091,Z 935.064,A -85,B 0,C 180,E1 10118.586,E2 10118.586} C_VEL
LIN {X 0,Y 271.454,Z 929.093,A -85,B 0,C 180,E1 10117.572,E2 10117.572} C_VEL
LIN {X 0,Y 271.811,Z 915.608,A -85,B 0,C 180,E1 10115.094,E2 10115.094} C_VEL
LIN {X 0,Y 272.499,Z 909.089,A -85,B 0,C 180,E1 10114.223,E2 10114.223} C_VEL
LIN {X 0,Y 272.888,Z 907.114,A -85,B 0,C 180,E1 10114.029,E2 10114.029} C_VEL
LIN {X 0,Y 276.338,Z 890.399,A -85,B 0,C 180,E1 10112.729,E2 10112.729} C_VEL
LIN {X 0,Y 278.806,Z 873.317,A -85,B 0,C 180,E1 10111.772,E2 10111.772} C_VEL
LIN {X 0,Y 280.266,Z 855.272,A -85,B 0,C 180,E1 10111.119,E2 10111.119} C_VEL
LIN {X 0,Y 286.891,Z 757.155,A -85,B 0,C 180,E1 10108.677,E2 10108.677} C_VEL
LIN {X 0,Y 285.93,Z 751.194,A -85,B 0,C 180,E1 10108.141,E2 10108.141} C_VEL
LIN {X 0,Y 280.041,Z 739.666,A -85,B 0,C 180,E1 10105.823,E2 10105.823} C_VEL
LIN {X 0,Y 273.976,Z 729.276,A -85,B 0,C 180,E1 10103.213,E2 10103.213} C_VEL
LIN {X 0,Y 268.318,Z 720.083,A -85,B 0,C 180,E1 10100.448,E2 10100.448} C_VEL
LIN {X 0,Y 263.26,Z 712.795,A -85,B 0,C 180,E1 10097.632,E2 10097.632} C_VEL
LIN {X 0,Y 258.508,Z 706.222,A -85,B 0,C 180,E1 10094.561,E2 10094.561} C_VEL
LIN {X 0,Y 254.126,Z 700.174,A -85,B 0,C 180,E1 10090.887,E2 10090.887} C_VEL
LIN {X 0,Y 253.435,Z 698.158,A -85,B 0,C 180,E1 10088.851,E2 10088.851} C_VEL
LIN {X 0,Y 252.581,Z 695.213,A -85,B 0,C 180,E1 10084.997,E2 10084.997} C_VEL
LIN {X 0,Y 251.807,Z 692.236,A -85,B 0,C 180,E1 10077.952,E2 10077.952} C_VEL
LIN {X 0,Y 252.07,Z 692.325,A -85,B 0,C 180,E1 10072.708,E2 10072.708} C_VEL
LIN {X 0,Y 252.495,Z 693.59,A -85,B 0,C 180,E1 10069.128,E2 10069.128} C_VEL
LIN {X 0,Y 254.375,Z 697.334,A -85,B 0,C 180,E1 10063.09,E2 10063.09} C_VEL
LIN {X 0,Y 256.155,Z 701.617,A -85,B 0,C 180,E1 10058.89,E2 10058.89} C_VEL
LIN {X 0,Y 257.642,Z 704.357,A -85,B 0,C 180,E1 10057.045,E2 10057.045} C_VEL
LIN {X 0,Y 263.019,Z 711.467,A -85,B 0,C 180,E1 10053.531,E2 10053.531} C_VEL
LIN {X 0,Y 268.312,Z 718.993,A -85,B 0,C 180,E1 10050.596,E2 10050.596} C_VEL
LIN {X 0,Y 273.298,Z 726.596,A -85,B 0,C 180,E1 10048.148,E2 10048.148} C_VEL
LIN {X 0,Y 279.43,Z 736.562,A -85,B 0,C 180,E1 10045.48,E2 10045.48} C_VEL
LIN {X 0,Y 285.992,Z 748.72,A -85,B 0,C 180,E1 10042.91,E2 10042.91} C_VEL
LIN {X 0,Y 287.038,Z 751.162,A -85,B 0,C 180,E1 10042.503,E2 10042.503} C_VEL
LIN {X 0,Y 287.377,Z 763.279,A -85,B 0,C 180,E1 10041.882,E2 10041.882} C_VEL
LIN {X 0,Y 278.146,Z 899.646,A -85,B 0,C 180,E1 10038.547,E2 10038.547} C_VEL
LIN {X 0,Y 275.558,Z 918.34,A -85,B 0,C 180,E1 10037.818,E2 10037.818} C_VEL
LIN {X 0,Y 271.844,Z 936.31,A -85,B 0,C 180,E1 10036.822,E2 10036.822} C_VEL
LIN {X 0,Y 267.22,Z 953.729,A -85,B 0,C 180,E1 10035.494,E2 10035.494} C_VEL
LIN {X 0,Y 262.06,Z 970.046,A -85,B 0,C 180,E1 10033.842,E2 10033.842} C_VEL
LIN {X 0,Y 256.45,Z 985.558,A -85,B 0,C 180,E1 10031.812,E2 10031.812} C_VEL
LIN {X 0,Y 250.6,Z 1000.173,A -85,B 0,C 180,E1 10029.374,E2 10029.374} C_VEL
LIN {X 0,Y 244.913,Z 1013.423,A -85,B 0,C 180,E1 10026.587,E2 10026.587} C_VEL
LIN {X 0,Y 239.206,Z 1026.226,A -85,B 0,C 180,E1 10023.2,E2 10023.2} C_VEL
LIN {X 0,Y 234.191,Z 1037.534,A -85,B 0,C 180,E1 10019.405,E2 10019.405} C_VEL
LIN {X 0,Y 230.094,Z 1047.335,A -85,B 0,C 180,E1 10015.204,E2 10015.204} C_VEL
LIN {X 0,Y 227.128,Z 1055.615,A -85,B 0,C 180,E1 10010.62,E2 10010.62} C_VEL
LIN {X 0,Y 225.516,Z 1062.141,A -85,B 0,C 180,E1 10005.826,E2 10005.826} C_VEL
LIN {X 0,Y 225.161,Z 1066.793,A -85,B 0,C 180,E1 10001.007,E2 10001.007} C_VEL
LIN {X 0,Y 225.697,Z 1069.565,A -85,B 0,C 180,E1 9996.358,E2 9996.358} C_VEL
LIN {X 0,Y 226.407,Z 1070.56,A -85,B 0,C 180,E1 9992.277,E2 9992.277} C_VEL
LIN {X 0,Y 226.608,Z 1070.192,A -85,B 0,C 180,E1 9988.988,E2 9988.988} C_VEL
LIN {X 0,Y 226.188,Z 1068.507,A -85,B 0,C 180,E1 9985.181,E2 9985.181} C_VEL
LIN {X 0,Y 225.48,Z 1065.704,A -85,B 0,C 180,E1 9980.556,E2 9980.556} C_VEL
LIN {X 0,Y 225.43,Z 1061.186,A -85,B 0,C 180,E1 9976.248,E2 9976.248} C_VEL
LIN {X 0,Y 226.271,Z 1054.801,A -85,B 0,C 180,E1 9971.981,E2 9971.981} C_VEL
LIN {X 0,Y 228.076,Z 1046.524,A -85,B 0,C 180,E1 9967.85,E2 9967.85} C_VEL
LIN {X 0,Y 230.722,Z 1036.826,A -85,B 0,C 180,E1 9964.042,E2 9964.042} C_VEL
LIN {X 0,Y 233.999,Z 1025.769,A -85,B 0,C 180,E1 9960.568,E2 9960.568} C_VEL
LIN {X 0,Y 238.126,Z 1012.389,A -85,B 0,C 180,E1 9957.203,E2 9957.203} C_VEL
LIN {X 0,Y 242.497,Z 997.902,A -85,B 0,C 180,E1 9954.317,E2 9954.317} C_VEL
LIN {X 0,Y 246.841,Z 982.414,A -85,B 0,C 180,E1 9951.849,E2 9951.849} C_VEL
LIN {X 0,Y 250.924,Z 965.915,A -85,B 0,C 180,E1 9949.794,E2 9949.794} C_VEL
LIN {X 0,Y 254.393,Z 949.62,A -85,B 0,C 180,E1 9948.225,E2 9948.225} C_VEL
LIN {X 0,Y 257.39,Z 931.492,A -85,B 0,C 180,E1 9946.962,E2 9946.962} C_VEL
LIN {X 0,Y 262.794,Z 887.377,A -85,B 0,C 180,E1 9944.943,E2 9944.943} C_VEL
LIN {X 0,Y 277.57,Z 782.86,A -85,B 0,C 180,E1 9940.875,E2 9940.875} C_VEL
LIN {X 0,Y 278.922,Z 775.027,A -85,B 0,C 180,E1 9940.538,E2 9940.538} C_VEL
LIN {X 0,Y 282.756,Z 761.695,A -85,B 0,C 180,E1 9939.725,E2 9939.725} C_VEL
LIN {X 0,Y 287.505,Z 744.525,A -85,B 0,C 180,E1 9938.131,E2 9938.131} C_VEL
LIN {X 0,Y 288.928,Z 735.519,A -85,B 0,C 180,E1 9935.243,E2 9935.243} C_VEL
LIN {X 0,Y 290.071,Z 731.526,A -85,B 0,C 180,E1 9933.708,E2 9933.708} C_VEL
LIN {X 0,Y 289.582,Z 732.552,A -85,B 0,C 180,E1 9931.656,E2 9931.656} C_VEL
LIN {X 0,Y 289.103,Z 735.531,A -85,B 0,C 180,E1 9929.186,E2 9929.186} C_VEL
LIN {X 0,Y 288.923,Z 739.894,A -85,B 0,C 180,E1 9926.736,E2 9926.736} C_VEL
LIN {X 0,Y 288.674,Z 745.938,A -85,B 0,C 180,E1 9924.341,E2 9924.341} C_VEL
LIN {X 0,Y 288.354,Z 749.165,A -85,B 0,C 180,E1 9923.392,E2 9923.392} C_VEL
LIN {X 0,Y 286.57,Z 756.971,A -85,B 0,C 180,E1 9922.19,E2 9922.19} C_VEL
LIN {X 0,Y 286.667,Z 763.118,A -85,B 0,C 180,E1 9921.489,E2 9921.489} C_VEL
LIN {X 0,Y 273.217,Z 866.008,A -85,B 0,C 180,E1 9917.765,E2 9917.765} C_VEL
LIN {X 0,Y 270.219,Z 896.233,A -85,B 0,C 180,E1 9916.325,E2 9916.325} C_VEL
LIN {X 0,Y 268.047,Z 911.675,A -85,B 0,C 180,E1 9915.246,E2 9915.246} C_VEL
LIN {X 0,Y 265.098,Z 926.585,A -85,B 0,C 180,E1 9913.857,E2 9913.857} C_VEL
LIN {X 0,Y 261.041,Z 942.135,A -85,B 0,C 180,E1 9911.937,E2 9911.937} C_VEL
LIN {X 0,Y 256.855,Z 955.044,A -85,B 0,C 180,E1 9909.862,E2 9909.862} C_VEL
LIN {X 0,Y 252.476,Z 966.62,A -85,B 0,C 180,E1 9907.509,E2 9907.509} C_VEL
LIN {X 0,Y 247.621,Z 977.529,A -85,B 0,C 180,E1 9904.632,E2 9904.632} C_VEL
LIN {X 0,Y 243.227,Z 986.211,A -85,B 0,C 180,E1 9901.649,E2 9901.649} C_VEL
LIN {X 0,Y 238.778,Z 993.899,A -85,B 0,C 180,E1 9898.08,E2 9898.08} C_VEL
LIN {X 0,Y 235.272,Z 999.118,A -85,B 0,C 180,E1 9894.635,E2 9894.635} C_VEL
LIN {X 0,Y 232.073,Z 1003.055,A -85,B 0,C 180,E1 9890.577,E2 9890.577} C_VEL
LIN {X 0,Y 229.822,Z 1004.836,A -85,B 0,C 180,E1 9886.668,E2 9886.668} C_VEL
LIN {X 0,Y 228.302,Z 1004.865,A -85,B 0,C 180,E1 9882.673,E2 9882.673} C_VEL
LIN {X 0,Y 227.461,Z 1003.123,A -85,B 0,C 180,E1 9878.734,E2 9878.734} C_VEL
LIN {X 0,Y 227.19,Z 999.591,A -85,B 0,C 180,E1 9874.729,E2 9874.729} C_VEL
LIN {X 0,Y 227.471,Z 994.246,A -85,B 0,C 180,E1 9870.796,E2 9870.796} C_VEL
LIN {X 0,Y 228.262,Z 987.355,A -85,B 0,C 180,E1 9867.1,E2 9867.1} C_VEL
LIN {X 0,Y 229.48,Z 978.95,A -85,B 0,C 180,E1 9863.66,E2 9863.66} C_VEL
LIN {X 0,Y 231.143,Z 968.733,A -85,B 0,C 180,E1 9860.353,E2 9860.353} C_VEL
LIN {X 0,Y 233.099,Z 956.912,A -85,B 0,C 180,E1 9857.333,E2 9857.333} C_VEL
LIN {X 0,Y 235.191,Z 943.836,A -85,B 0,C 180,E1 9854.663,E2 9854.663} C_VEL
LIN {X 0,Y 237.278,Z 929.345,A -85,B 0,C 180,E1 9852.325,E2 9852.325} C_VEL
LIN {X 0,Y 239.159,Z 913.947,A -85,B 0,C 180,E1 9850.393,E2 9850.393} C_VEL
LIN {X 0,Y 240.718,Z 897.72,A -85,B 0,C 180,E1 9848.845,E2 9848.845} C_VEL
LIN {X 0,Y 241.908,Z 879.254,A -85,B 0,C 180,E1 9847.614,E2 9847.614} C_VEL
LIN {X 0,Y 243.893,Z 830.171,A -85,B 0,C 180,E1 9845.666,E2 9845.666} C_VEL
LIN {X 0,Y 249.161,Z 741.121,A -85,B 0,C 180,E1 9842.445,E2 9842.445} C_VEL
LIN {X 0,Y 248.274,Z 732.433,A -85,B 0,C 180,E1 9841.91,E2 9841.91} C_VEL
LIN {X 0,Y 249.98,Z 712.948,A -85,B 0,C 180,E1 9838.946,E2 9838.946} C_VEL
LIN {X 0,Y 248.242,Z 705.425,A -85,B 0,C 180,E1 9837.334,E2 9837.334} C_VEL
LIN {X 0,Y 248.827,Z 704.983,A -85,B 0,C 180,E1 9836.865,E2 9836.865} C_VEL
LIN {X 0,Y 249.677,Z 705.553,A -85,B 0,C 180,E1 9836.628,E2 9836.628} C_VEL
LIN {X 0,Y 257.568,Z 721.023,A -85,B 0,C 180,E1 9834.484,E2 9834.484} C_VEL
LIN {X 0,Y 259.709,Z 726.166,A -85,B 0,C 180,E1 9833.901,E2 9833.901} C_VEL
LIN {X 0,Y 263.041,Z 750.058,A -85,B 0,C 180,E1 9832.476,E2 9832.476} C_VEL
LIN {X 0,Y 257.503,Z 859.568,A -85,B 0,C 180,E1 9829.567,E2 9829.567} C_VEL
LIN {X 0,Y 256.185,Z 877.029,A -85,B 0,C 180,E1 9828.747,E2 9828.747} C_VEL
LIN {X 0,Y 254.241,Z 893.047,A -85,B 0,C 180,E1 9827.628,E2 9827.628} C_VEL
LIN {X 0,Y 251.492,Z 909.74,A -85,B 0,C 180,E1 9826.041,E2 9826.041} C_VEL
LIN {X 0,Y 248.303,Z 925.271,A -85,B 0,C 180,E1 9824.101,E2 9824.101} C_VEL
LIN {X 0,Y 244.791,Z 939.608,A -85,B 0,C 180,E1 9821.785,E2 9821.785} C_VEL
LIN {X 0,Y 241.14,Z 952.907,A -85,B 0,C 180,E1 9819.066,E2 9819.066} C_VEL
LIN {X 0,Y 237.637,Z 964.664,A -85,B 0,C 180,E1 9816.039,E2 9816.039} C_VEL
LIN {X 0,Y 234.411,Z 974.88,A -85,B 0,C 180,E1 9812.69,E2 9812.69} C_VEL
LIN {X 0,Y 231.644,Z 983.667,A -85,B 0,C 180,E1 9809.011,E2 9809.011} C_VEL
LIN {X 0,Y 229.474,Z 990.995,A -85,B 0,C 180,E1 9805.001,E2 9805.001} C_VEL
LIN {X 0,Y 228.072,Z 996.42,A -85,B 0,C 180,E1 9800.92,E2 9800.92} C_VEL
LIN {X 0,Y 227.338,Z 1000.331,A -85,B 0,C 180,E1 9796.521,E2 9796.521} C_VEL
LIN {X 0,Y 227.355,Z 1002.493,A -85,B 0,C 180,E1 9792.071,E2 9792.071} C_VEL
LIN {X 0,Y 228.147,Z 1002.905,A -85,B 0,C 180,E1 9787.588,E2 9787.588} C_VEL
LIN {X 0,Y 229.818,Z 1001.476,A -85,B 0,C 180,E1 9783.099,E2 9783.099} C_VEL
LIN {X 0,Y 232.309,Z 998.426,A -85,B 0,C 180,E1 9778.904,E2 9778.904} C_VEL
LIN {X 0,Y 235.785,Z 993.568,A -85,B 0,C 180,E1 9774.781,E2 9774.781} C_VEL
LIN {X 0,Y 239.946,Z 987.107,A -85,B 0,C 180,E1 9771.008,E2 9771.008} C_VEL
LIN {X 0,Y 244.98,Z 978.587,A -85,B 0,C 180,E1 9767.351,E2 9767.351} C_VEL
LIN {X 0,Y 250.015,Z 969.235,A -85,B 0,C 180,E1 9764.287,E2 9764.287} C_VEL
LIN {X 0,Y 255.488,Z 957.932,A -85,B 0,C 180,E1 9761.406,E2 9761.406} C_VEL
LIN {X 0,Y 260.831,Z 945.295,A -85,B 0,C 180,E1 9758.907,E2 9758.907} C_VEL
LIN {X 0,Y 266.046,Z 931.023,A -85,B 0,C 180,E1 9756.696,E2 9756.696} C_VEL
LIN {X 0,Y 270.621,Z 916.047,A -85,B 0,C 180,E1 9754.894,E2 9754.894} C_VEL
LIN {X 0,Y 272.888,Z 907.114,A -85,B 0,C 180,E1 9754.029,E2 9754.029} C_VEL
LIN {X 0,Y 273.84,Z 900.247,A -85,B 0,C 180,E1 9753.288,E2 9753.288} C_VEL
LIN {X 0,Y 273.258,Z 884.038,A -85,B 0,C 180,E1 9751.218,E2 9751.218} C_VEL
LIN {X 0,Y 273.506,Z 876.854,A -85,B 0,C 180,E1 9750.62,E2 9750.62} C_VEL
LIN {X 0,Y 273.625,Z 875.79,A -85,B 0,C 180,E1 9750.563,E2 9750.563} C_VEL
LIN {X 0,Y 275.252,Z 858.16,A -85,B 0,C 180,E1 9749.884,E2 9749.884} C_VEL
LIN {X 0,Y 282.205,Z 758.963,A -85,B 0,C 180,E1 9747.397,E2 9747.397} C_VEL
LIN {X 0,Y 281.603,Z 755.594,A -85,B 0,C 180,E1 9747.06,E2 9747.06} C_VEL
LIN {X 0,Y 275.224,Z 743.04,A -85,B 0,C 180,E1 9744.381,E2 9744.381} C_VEL
LIN {X 0,Y 268.771,Z 731.805,A -85,B 0,C 180,E1 9741.324,E2 9741.324} C_VEL
LIN {X 0,Y 264.082,Z 724.552,A -85,B 0,C 180,E1 9738.825,E2 9738.825} C_VEL
LIN {X 0,Y 260.922,Z 719.773,A -85,B 0,C 180,E1 9736.932,E2 9736.932} C_VEL
LIN {X 0,Y 256.557,Z 713.558,A -85,B 0,C 180,E1 9733.983,E2 9733.983} C_VEL
LIN {X 0,Y 251.464,Z 706.538,A -85,B 0,C 180,E1 9729.614,E2 9729.614} C_VEL
LIN {X 0,Y 247.573,Z 701.431,A -85,B 0,C 180,E1 9724.866,E2 9724.866} C_VEL
LIN {X 0,Y 246.63,Z 698.783,A -85,B 0,C 180,E1 9719.304,E2 9719.304} C_VEL
LIN {X 0,Y 246.714,Z 698.262,A -85,B 0,C 180,E1 9715.817,E2 9715.817} C_VEL
LIN {X 0,Y 247.189,Z 698.861,A -85,B 0,C 180,E1 9711.159,E2 9711.159} C_VEL
LIN {X 0,Y 248.86,Z 702.595,A -85,B 0,C 180,E1 9704.384,E2 9704.384} C_VEL
LIN {X 0,Y 250.945,Z 705.714,A -85,B 0,C 180,E1 9701.894,E2 9701.894} C_VEL
LIN {X 0,Y 254.307,Z 709.792,A -85,B 0,C 180,E1 9698.795,E2 9698.795} C_VEL
LIN {X 0,Y 257.652,Z 714.47,A -85,B 0,C 180,E1 9696.198,E2 9696.198} C_VEL
LIN {X 0,Y 260.976,Z 718.888,A -85,B 0,C 180,E1 9694.042,E2 9694.042} C_VEL
LIN {X 0,Y 265.961,Z 726.209,A -85,B 0,C 180,E1 9691.171,E2 9691.171} C_VEL
LIN {X 0,Y 270.623,Z 733.516,A -85,B 0,C 180,E1 9688.79,E2 9688.79} C_VEL
LIN {X 0,Y 276.297,Z 743.107,A -85,B 0,C 180,E1 9686.194,E2 9686.194} C_VEL
LIN {X 0,Y 282.496,Z 754.915,A -85,B 0,C 180,E1 9683.657,E2 9683.657} C_VEL
LIN {X 0,Y 282.667,Z 764.524,A -85,B 0,C 180,E1 9683.169,E2 9683.169} C_VEL
LIN {X 0,Y 273.196,Z 898.827,A -85,B 0,C 180,E1 9679.868,E2 9679.868} C_VEL
LIN {X 0,Y 270.518,Z 917.495,A -85,B 0,C 180,E1 9679.138,E2 9679.138} C_VEL
LIN {X 0,Y 266.569,Z 935.87,A -85,B 0,C 180,E1 9678.114,E2 9678.114} C_VEL
LIN {X 0,Y 261.89,Z 952.791,A -85,B 0,C 180,E1 9676.82,E2 9676.82} C_VEL
LIN {X 0,Y 256.562,Z 968.983,A -85,B 0,C 180,E1 9675.176,E2 9675.176} C_VEL
LIN {X 0,Y 250.648,Z 984.662,A -85,B 0,C 180,E1 9673.114,E2 9673.114} C_VEL
LIN {X 0,Y 244.363,Z 999.622,A -85,B 0,C 180,E1 9670.585,E2 9670.585} C_VEL
LIN {X 0,Y 237.974,Z 1013.728,A -85,B 0,C 180,E1 9667.533,E2 9667.533} C_VEL
LIN {X 0,Y 232.018,Z 1026.239,A -85,B 0,C 180,E1 9664.07,E2 9664.07} C_VEL
LIN {X 0,Y 226.765,Z 1037.29,A -85,B 0,C 180,E1 9660.175,E2 9660.175} C_VEL
LIN {X 0,Y 222.452,Z 1046.898,A -85,B 0,C 180,E1 9655.847,E2 9655.847} C_VEL
LIN {X 0,Y 219.31,Z 1055.007,A -85,B 0,C 180,E1 9651.11,E2 9651.11} C_VEL
LIN {X 0,Y 217.559,Z 1061.519,A -85,B 0,C 180,E1 9646.006,E2 9646.006} C_VEL
LIN {X 0,Y 217.205,Z 1066.069,A -85,B 0,C 180,E1 9640.878,E2 9640.878} C_VEL
LIN {X 0,Y 217.763,Z 1068.497,A -85,B 0,C 180,E1 9636.326,E2 9636.326} C_VEL
LIN {X 0,Y 218.482,Z 1069.341,A -85,B 0,C 180,E1 9632.36,E2 9632.36} C_VEL
LIN {X 0,Y 218.7,Z 1068.944,A -85,B 0,C 180,E1 9628.951,E2 9628.951} C_VEL
LIN {X 0,Y 218.234,Z 1067.192,A -85,B 0,C 180,E1 9625.005,E2 9625.005} C_VEL
LIN {X 0,Y 217.507,Z 1064.809,A -85,B 0,C 180,E1 9620.474,E2 9620.474} C_VEL
LIN {X 0,Y 217.466,Z 1060.516,A -85,B 0,C 180,E1 9615.895,E2 9615.895} C_VEL
LIN {X 0,Y 218.461,Z 1054.121,A -85,B 0,C 180,E1 9611.313,E2 9611.313} C_VEL
LIN {X 0,Y 220.528,Z 1046.05,A -85,B 0,C 180,E1 9606.982,E2 9606.982} C_VEL
LIN {X 0,Y 223.665,Z 1035.984,A -85,B 0,C 180,E1 9602.822,E2 9602.822} C_VEL
LIN {X 0,Y 227.572,Z 1024.495,A -85,B 0,C 180,E1 9599.065,E2 9599.065} C_VEL
LIN {X 0,Y 232.537,Z 1010.28,A -85,B 0,C 180,E1 9595.418,E2 9595.418} C_VEL
LIN {X 0,Y 237.656,Z 995.177,A -85,B 0,C 180,E1 9592.407,E2 9592.407} C_VEL
LIN {X 0,Y 242.451,Z 979.724,A -85,B 0,C 180,E1 9589.958,E2 9589.958} C_VEL
LIN {X 0,Y 246.994,Z 963.239,A -85,B 0,C 180,E1 9587.935,E2 9587.935} C_VEL
LIN {X 0,Y 250.841,Z 946.899,A -85,B 0,C 180,E1 9586.402,E2 9586.402} C_VEL
LIN {X 0,Y 254.23,Z 928.547,A -85,B 0,C 180,E1 9585.172,E2 9585.172} C_VEL
LIN {X 0,Y 259.993,Z 885.735,A -85,B 0,C 180,E1 9583.246,E2 9583.246} C_VEL
LIN {X 0,Y 275.426,Z 783.894,A -85,B 0,C 180,E1 9579.292,E2 9579.292} C_VEL
LIN {X 0,Y 277.204,Z 773.338,A -85,B 0,C 180,E1 9578.821,E2 9578.821} C_VEL
LIN {X 0,Y 280.135,Z 763.992,A -85,B 0,C 180,E1 9578.258,E2 9578.258} C_VEL
LIN {X 0,Y 284.53,Z 749.14,A -85,B 0,C 180,E1 9576.846,E2 9576.846} C_VEL
LIN {X 0,Y 286.059,Z 741.761,A -85,B 0,C 180,E1 9574.422,E2 9574.422} C_VEL
LIN {X 0,Y 286.862,Z 739.098,A -85,B 0,C 180,E1 9573.415,E2 9573.415} C_VEL
LIN {X 0,Y 286.424,Z 739.945,A -85,B 0,C 180,E1 9571.81,E2 9571.81} C_VEL
LIN {X 0,Y 285.799,Z 742.807,A -85,B 0,C 180,E1 9569.41,E2 9569.41} C_VEL
LIN {X 0,Y 285.378,Z 746.925,A -85,B 0,C 180,E1 9567.095,E2 9567.095} C_VEL
LIN {X 0,Y 284.808,Z 753.103,A -85,B 0,C 180,E1 9564.693,E2 9564.693} C_VEL
LIN {X 0,Y 284.365,Z 755.047,A -85,B 0,C 180,E1 9564.291,E2 9564.291} C_VEL
LIN {X 0,Y 283.558,Z 759.175,A -85,B 0,C 180,E1 9563.674,E2 9563.674} C_VEL
LIN {X 0,Y 283.453,Z 765.549,A -85,B 0,C 180,E1 9562.918,E2 9562.918} C_VEL
LIN {X 0,Y 269.378,Z 866.981,A -85,B 0,C 180,E1 9559.233,E2 9559.233} C_VEL
LIN {X 0,Y 266.025,Z 897.584,A -85,B 0,C 180,E1 9557.752,E2 9557.752} C_VEL
LIN {X 0,Y 263.63,Z 913.333,A -85,B 0,C 180,E1 9556.639,E2 9556.639} C_VEL
LIN {X 0,Y 260.468,Z 928.086,A -85,B 0,C 180,E1 9555.245,E2 9555.245} C_VEL
LIN {X 0,Y 256.36,Z 942.819,A -85,B 0,C 180,E1 9553.418,E2 9553.418} C_VEL
LIN {X 0,Y 251.874,Z 955.873,A -85,B 0,C 180,E1 9551.327,E2 9551.327} C_VEL
LIN {X 0,Y 246.873,Z 968.181,A -85,B 0,C 180,E1 9548.797,E2 9548.797} C_VEL
LIN {X 0,Y 241.76,Z 978.859,A -85,B 0,C 180,E1 9545.934,E2 9545.934} C_VEL
LIN {X 0,Y 237.023,Z 987.537,A -85,B 0,C 180,E1 9542.901,E2 9542.901} C_VEL
LIN {X 0,Y 232.486,Z 994.756,A -85,B 0,C 180,E1 9539.507,E2 9539.507} C_VEL
LIN {X 0,Y 228.552,Z 1000.25,A -85,B 0,C 180,E1 9535.914,E2 9535.914} C_VEL
LIN {X 0,Y 225.162,Z 1004.07,A -85,B 0,C 180,E1 9532.001,E2 9532.001} C_VEL
LIN {X 0,Y 222.627,Z 1006.084,A -85,B 0,C 180,E1 9528.077,E2 9528.077} C_VEL
LIN {X 0,Y 220.736,Z 1006.318,A -85,B 0,C 180,E1 9523.802,E2 9523.802} C_VEL
LIN {X 0,Y 219.675,Z 1004.769,A -85,B 0,C 180,E1 9519.657,E2 9519.657} C_VEL
LIN {X 0,Y 219.253,Z 1001.355,A -85,B 0,C 180,E1 9515.481,E2 9515.481} C_VEL
LIN {X 0,Y 219.433,Z 996.241,A -85,B 0,C 180,E1 9511.416,E2 9511.416} C_VEL
LIN {X 0,Y 220.224,Z 988.945,A -85,B 0,C 180,E1 9507.296,E2 9507.296} C_VEL
LIN {X 0,Y 221.441,Z 980.66,A -85,B 0,C 180,E1 9503.736,E2 9503.736} C_VEL
LIN {X 0,Y 223.203,Z 970.075,A -85,B 0,C 180,E1 9500.164,E2 9500.164} C_VEL
LIN {X 0,Y 225.168,Z 958.57,A -85,B 0,C 180,E1 9497.113,E2 9497.113} C_VEL
LIN {X 0,Y 227.292,Z 945.764,A -85,B 0,C 180,E1 9494.383,E2 9494.383} C_VEL
LIN {X 0,Y 229.551,Z 930.639,A -85,B 0,C 180,E1 9491.855,E2 9491.855} C_VEL
LIN {X 0,Y 231.514,Z 915.154,A -85,B 0,C 180,E1 9489.849,E2 9489.849} C_VEL
LIN {X 0,Y 233.107,Z 899.312,A -85,B 0,C 180,E1 9488.284,E2 9488.284} C_VEL
LIN {X 0,Y 234.352,Z 881.101,A -85,B 0,C 180,E1 9487.019,E2 9487.019} C_VEL
LIN {X 0,Y 235.776,Z 843.794,A -85,B 0,C 180,E1 9485.443,E2 9485.443} C_VEL
LIN {X 0,Y 242.005,Z 742.083,A -85,B 0,C 180,E1 9481.623,E2 9481.623} C_VEL
LIN {X 0,Y 241.155,Z 733.523,A -85,B 0,C 180,E1 9481.088,E2 9481.088} C_VEL
LIN {X 0,Y 242.875,Z 715.406,A -85,B 0,C 180,E1 9478.237,E2 9478.237} C_VEL
LIN {X 0,Y 243.068,Z 714.604,A -85,B 0,C 180,E1 9477.821,E2 9477.821} C_VEL
LIN {X 0,Y 245.64,Z 714.832,A -85,B 0,C 180,E1 9477.123,E2 9477.123} C_VEL
LIN {X 0,Y 246.867,Z 714.707,A -85,B 0,C 180,E1 9476.866,E2 9476.866} C_VEL
LIN {X 0,Y 253.799,Z 729.248,A -85,B 0,C 180,E1 9474.907,E2 9474.907} C_VEL
LIN {X 0,Y 256.741,Z 751.329,A -85,B 0,C 180,E1 9473.55,E2 9473.55} C_VEL
LIN {X 0,Y 251.006,Z 860.104,A -85,B 0,C 180,E1 9470.612,E2 9470.612} C_VEL
LIN {X 0,Y 249.629,Z 877.665,A -85,B 0,C 180,E1 9469.776,E2 9469.776} C_VEL
LIN {X 0,Y 247.553,Z 894.042,A -85,B 0,C 180,E1 9468.608,E2 9468.608} C_VEL
LIN {X 0,Y 244.688,Z 910.709,A -85,B 0,C 180,E1 9466.988,E2 9466.988} C_VEL
LIN {X 0,Y 241.363,Z 926.226,A -85,B 0,C 180,E1 9465.006,E2 9465.006} C_VEL
LIN {X 0,Y 237.701,Z 940.565,A -85,B 0,C 180,E1 9462.635,E2 9462.635} C_VEL
LIN {X 0,Y 233.887,Z 953.875,A -85,B 0,C 180,E1 9459.847,E2 9459.847} C_VEL
LIN {X 0,Y 230.224,Z 965.649,A -85,B 0,C 180,E1 9456.735,E2 9456.735} C_VEL
LIN {X 0,Y 226.845,Z 975.887,A -85,B 0,C 180,E1 9453.286,E2 9453.286} C_VEL
LIN {X 0,Y 223.94,Z 984.697,A -85,B 0,C 180,E1 9449.489,E2 9449.489} C_VEL
LIN {X 0,Y 221.66,Z 992.053,A -85,B 0,C 180,E1 9445.343,E2 9445.343} C_VEL
LIN {X 0,Y 220.186,Z 997.519,A -85,B 0,C 180,E1 9441.119,E2 9441.119} C_VEL
LIN {X 0,Y 219.418,Z 1001.463,A -85,B 0,C 180,E1 9436.562,E2 9436.562} C_VEL
LIN {X 0,Y 219.447,Z 1003.664,A -85,B 0,C 180,E1 9431.952,E2 9431.952} C_VEL
LIN {X 0,Y 220.301,Z 1004.133,A -85,B 0,C 180,E1 9427.308,E2 9427.308} C_VEL
LIN {X 0,Y 222.086,Z 1002.751,A -85,B 0,C 180,E1 9422.664,E2 9422.664} C_VEL
LIN {X 0,Y 224.935,Z 999.515,A -85,B 0,C 180,E1 9418.065,E2 9418.065} C_VEL
LIN {X 0,Y 228.676,Z 994.598,A -85,B 0,C 180,E1 9413.824,E2 9413.824} C_VEL
LIN {X 0,Y 233.117,Z 988.079,A -85,B 0,C 180,E1 9409.958,E2 9409.958} C_VEL
LIN {X 0,Y 238.455,Z 979.515,A -85,B 0,C 180,E1 9406.223,E2 9406.223} C_VEL
LIN {X 0,Y 243.77,Z 970.135,A -85,B 0,C 180,E1 9403.107,E2 9403.107} C_VEL
LIN {X 0,Y 249.549,Z 958.737,A -85,B 0,C 180,E1 9400.172,E2 9400.172} C_VEL
LIN {X 0,Y 255.121,Z 946.156,A -85,B 0,C 180,E1 9397.659,E2 9397.659} C_VEL
LIN {X 0,Y 260.376,Z 932.39,A -85,B 0,C 180,E1 9395.503,E2 9395.503} C_VEL
LIN {X 0,Y 265.232,Z 917.199,A -85,B 0,C 180,E1 9393.653,E2 9393.653} C_VEL
LIN {X 0,Y 269.295,Z 901.068,A -85,B 0,C 180,E1 9392.164,E2 9392.164} C_VEL
LIN {X 0,Y 272.509,Z 883.821,A -85,B 0,C 180,E1 9390.986,E2 9390.986} C_VEL
LIN {X 0,Y 273.625,Z 875.79,A -85,B 0,C 180,E1 9390.563,E2 9390.563} C_VEL
LIN {X 0,Y 273.864,Z 868.392,A -85,B 0,C 180,E1 9390.07,E2 9390.07} C_VEL
LIN {X 0,Y 271.68,Z 849.933,A -85,B 0,C 180,E1 9388.459,E2 9388.459} C_VEL
LIN {X 0,Y 271.62,Z 842.389,A -85,B 0,C 180,E1 9388.095,E2 9388.095} C_VEL
LIN {X 0,Y 277.644,Z 760.652,A -85,B 0,C 180,E1 9386.063,E2 9386.063} C_VEL
LIN {X 0,Y 271.744,Z 748.654,A -85,B 0,C 180,E1 9383.415,E2 9383.415} C_VEL
LIN {X 0,Y 265.657,Z 737.906,A -85,B 0,C 180,E1 9380.374,E2 9380.374} C_VEL
LIN {X 0,Y 261.689,Z 731.519,A -85,B 0,C 180,E1 9378.144,E2 9378.144} C_VEL
LIN {X 0,Y 258.383,Z 726.401,A -85,B 0,C 180,E1 9376.063,E2 9376.063} C_VEL
LIN {X 0,Y 254.655,Z 720.893,A -85,B 0,C 180,E1 9373.395,E2 9373.395} C_VEL
LIN {X 0,Y 249.886,Z 714.054,A -85,B 0,C 180,E1 9369.094,E2 9369.094} C_VEL
LIN {X 0,Y 246.245,Z 709.126,A -85,B 0,C 180,E1 9364.425,E2 9364.425} C_VEL
LIN {X 0,Y 243.661,Z 705.751,A -85,B 0,C 180,E1 9357.649,E2 9357.649} C_VEL
LIN {X 0,Y 243.88,Z 705.93,A -85,B 0,C 180,E1 9352.225,E2 9352.225} C_VEL
LIN {X 0,Y 245.711,Z 708.56,A -85,B 0,C 180,E1 9347.307,E2 9347.307} C_VEL
LIN {X 0,Y 248.171,Z 711.241,A -85,B 0,C 180,E1 9343.86,E2 9343.86} C_VEL
LIN {X 0,Y 253.037,Z 717.861,A -85,B 0,C 180,E1 9338.926,E2 9338.926} C_VEL
LIN {X 0,Y 258.473,Z 725.528,A -85,B 0,C 180,E1 9334.878,E2 9334.878} C_VEL
LIN {X 0,Y 263.538,Z 733.247,A -85,B 0,C 180,E1 9331.813,E2 9331.813} C_VEL
LIN {X 0,Y 267.982,Z 740.432,A -85,B 0,C 180,E1 9329.446,E2 9329.446} C_VEL
LIN {X 0,Y 273.267,Z 749.757,A -85,B 0,C 180,E1 9326.901,E2 9326.901} C_VEL
LIN {X 0,Y 278.092,Z 759.262,A -85,B 0,C 180,E1 9324.813,E2 9324.813} C_VEL
LIN {X 0,Y 278.096,Z 765.889,A -85,B 0,C 180,E1 9324.495,E2 9324.495} C_VEL
LIN {X 0,Y 268.406,Z 897.992,A -85,B 0,C 180,E1 9321.238,E2 9321.238} C_VEL
LIN {X 0,Y 265.639,Z 916.672,A -85,B 0,C 180,E1 9320.509,E2 9320.509} C_VEL
LIN {X 0,Y 261.635,Z 934.763,A -85,B 0,C 180,E1 9319.507,E2 9319.507} C_VEL
LIN {X 0,Y 256.778,Z 951.749,A -85,B 0,C 180,E1 9318.216,E2 9318.216} C_VEL
LIN {X 0,Y 251.243,Z 967.944,A -85,B 0,C 180,E1 9316.575,E2 9316.575} C_VEL
LIN {X 0,Y 245.175,Z 983.362,A -85,B 0,C 180,E1 9314.542,E2 9314.542} C_VEL
LIN {X 0,Y 238.751,Z 997.95,A -85,B 0,C 180,E1 9312.071,E2 9312.071} C_VEL
LIN {X 0,Y 232.45,Z 1011.183,A -85,B 0,C 180,E1 9309.22,E2 9309.22} C_VEL
LIN {X 0,Y 226.049,Z 1023.954,A -85,B 0,C 180,E1 9305.722,E2 9305.722} C_VEL
LIN {X 0,Y 220.326,Z 1035.222,A -85,B 0,C 180,E1 9301.763,E2 9301.763} C_VEL
LIN {X 0,Y 215.544,Z 1044.978,A -85,B 0,C 180,E1 9297.337,E2 9297.337} C_VEL
LIN {X 0,Y 211.958,Z 1053.228,A -85,B 0,C 180,E1 9292.463,E2 9292.463} C_VEL
LIN {X 0,Y 209.898,Z 1059.581,A -85,B 0,C 180,E1 9287.463,E2 9287.463} C_VEL
LIN {X 0,Y 209.207,Z 1064.357,A -85,B 0,C 180,E1 9282.139,E2 9282.139} C_VEL
LIN {X 0,Y 209.683,Z 1067.126,A -85,B 0,C 180,E1 9277.121,E2 9277.121} C_VEL
LIN {X 0,Y 210.51,Z 1068.121,A -85,B 0,C 180,E1 9272.722,E2 9272.722} C_VEL
LIN {X 0,Y 210.805,Z 1067.76,A -85,B 0,C 180,E1 9269.184,E2 9269.184} C_VEL
LIN {X 0,Y 210.368,Z 1066.189,A -85,B 0,C 180,E1 9265.365,E2 9265.365} C_VEL
LIN {X 0,Y 209.532,Z 1063.916,A -85,B 0,C 180,E1 9260.385,E2 9260.385} C_VEL
LIN {X 0,Y 209.5,Z 1059.895,A -85,B 0,C 180,E1 9255.63,E2 9255.63} C_VEL
LIN {X 0,Y 210.484,Z 1054.343,A -85,B 0,C 180,E1 9251.154,E2 9251.154} C_VEL
LIN {X 0,Y 212.834,Z 1046.174,A -85,B 0,C 180,E1 9246.358,E2 9246.358} C_VEL
LIN {X 0,Y 216.391,Z 1036.167,A -85,B 0,C 180,E1 9241.88,E2 9241.88} C_VEL
LIN {X 0,Y 221.011,Z 1024.182,A -85,B 0,C 180,E1 9237.734,E2 9237.734} C_VEL
LIN {X 0,Y 226.048,Z 1011.397,A -85,B 0,C 180,E1 9234.276,E2 9234.276} C_VEL
LIN {X 0,Y 231.777,Z 996.543,A -85,B 0,C 180,E1 9231.121,E2 9231.121} C_VEL
LIN {X 0,Y 237.176,Z 981.117,A -85,B 0,C 180,E1 9228.557,E2 9228.557} C_VEL
LIN {X 0,Y 242.094,Z 965.724,A -85,B 0,C 180,E1 9226.554,E2 9226.554} C_VEL
LIN {X 0,Y 246.8,Z 948.341,A -85,B 0,C 180,E1 9224.847,E2 9224.847} C_VEL
LIN {X 0,Y 250.471,Z 931.443,A -85,B 0,C 180,E1 9223.652,E2 9223.652} C_VEL
LIN {X 0,Y 254.246,Z 906.883,A -85,B 0,C 180,E1 9222.439,E2 9222.439} C_VEL
LIN {X 0,Y 273.658,Z 784.89,A -85,B 0,C 180,E1 9217.675,E2 9217.675} C_VEL
LIN {X 0,Y 276.187,Z 771.063,A -85,B 0,C 180,E1 9217.035,E2 9217.035} C_VEL
LIN {X 0,Y 278.145,Z 764.965,A -85,B 0,C 180,E1 9216.635,E2 9216.635} C_VEL
LIN {X 0,Y 281.728,Z 753.977,A -85,B 0,C 180,E1 9215.594,E2 9215.594} C_VEL
LIN {X 0,Y 283.256,Z 748.01,A -85,B 0,C 180,E1 9213.586,E2 9213.586} C_VEL
LIN {X 0,Y 283.665,Z 746.674,A -85,B 0,C 180,E1 9212.975,E2 9212.975} C_VEL
LIN {X 0,Y 283.106,Z 747.816,A -85,B 0,C 180,E1 9211.513,E2 9211.513} C_VEL
LIN {X 0,Y 282.496,Z 750.331,A -85,B 0,C 180,E1 9209.46,E2 9209.46} C_VEL
LIN {X 0,Y 281.743,Z 755.058,A -85,B 0,C 180,E1 9207.016,E2 9207.016} C_VEL
LIN {X 0,Y 281.178,Z 758.944,A -85,B 0,C 180,E1 9205.551,E2 9205.551} C_VEL
LIN {X 0,Y 280.666,Z 768.01,A -85,B 0,C 180,E1 9204.394,E2 9204.394} C_VEL
LIN {X 0,Y 265.908,Z 867.91,A -85,B 0,C 180,E1 9200.763,E2 9200.763} C_VEL
LIN {X 0,Y 262.176,Z 898.903,A -85,B 0,C 180,E1 9199.247,E2 9199.247} C_VEL
LIN {X 0,Y 259.706,Z 914.149,A -85,B 0,C 180,E1 9198.17,E2 9198.17} C_VEL
LIN {X 0,Y 256.081,Z 929.859,A -85,B 0,C 180,E1 9196.677,E2 9196.677} C_VEL
LIN {X 0,Y 251.698,Z 944.456,A -85,B 0,C 180,E1 9194.846,E2 9194.846} C_VEL
LIN {X 0,Y 246.921,Z 957.403,A -85,B 0,C 180,E1 9192.749,E2 9192.749} C_VEL
LIN {X 0,Y 241.658,Z 969.42,A -85,B 0,C 180,E1 9190.248,E2 9190.248} C_VEL
LIN {X 0,Y 236.491,Z 979.549,A -85,B 0,C 180,E1 9187.531,E2 9187.531} C_VEL
LIN {X 0,Y 230.976,Z 988.952,A -85,B 0,C 180,E1 9184.22,E2 9184.22} C_VEL
LIN {X 0,Y 225.988,Z 996.238,A -85,B 0,C 180,E1 9180.704,E2 9180.704} C_VEL
LIN {X 0,Y 221.575,Z 1001.847,A -85,B 0,C 180,E1 9176.895,E2 9176.895} C_VEL
LIN {X 0,Y 217.687,Z 1005.767,A -85,B 0,C 180,E1 9172.61,E2 9172.61} C_VEL
LIN {X 0,Y 214.905,Z 1007.596,A -85,B 0,C 180,E1 9168.459,E2 9168.459} C_VEL
LIN {X 0,Y 212.844,Z 1007.595,A -85,B 0,C 180,E1 9163.909,E2 9163.909} C_VEL
LIN {X 0,Y 211.77,Z 1005.889,A -85,B 0,C 180,E1 9159.838,E2 9159.838} C_VEL
LIN {X 0,Y 211.304,Z 1002.124,A -85,B 0,C 180,E1 9155.303,E2 9155.303} C_VEL
LIN {X 0,Y 211.499,Z 996.845,A -85,B 0,C 180,E1 9151.17,E2 9151.17} C_VEL
LIN {X 0,Y 212.266,Z 989.92,A -85,B 0,C 180,E1 9147.2,E2 9147.2} C_VEL
LIN {X 0,Y 213.52,Z 981.514,A -85,B 0,C 180,E1 9143.507,E2 9143.507} C_VEL
LIN {X 0,Y 215.348,Z 970.791,A -85,B 0,C 180,E1 9139.805,E2 9139.805} C_VEL
LIN {X 0,Y 217.558,Z 958.23,A -85,B 0,C 180,E1 9136.419,E2 9136.419} C_VEL
LIN {X 0,Y 219.747,Z 945.32,A -85,B 0,C 180,E1 9133.659,E2 9133.659} C_VEL
LIN {X 0,Y 222.076,Z 930.181,A -85,B 0,C 180,E1 9131.098,E2 9131.098} C_VEL
LIN {X 0,Y 224.203,Z 913.659,A -85,B 0,C 180,E1 9128.963,E2 9128.963} C_VEL
LIN {X 0,Y 225.778,Z 897.786,A -85,B 0,C 180,E1 9127.43,E2 9127.43} C_VEL
LIN {X 0,Y 226.952,Z 880.566,A -85,B 0,C 180,E1 9126.247,E2 9126.247} C_VEL
LIN {X 0,Y 229.301,Z 828.899,A -85,B 0,C 180,E1 9124.069,E2 9124.069} C_VEL
LIN {X 0,Y 234.885,Z 742.932,A -85,B 0,C 180,E1 9120.748,E2 9120.748} C_VEL
LIN {X 0,Y 234.113,Z 734.538,A -85,B 0,C 180,E1 9120.196,E2 9120.196} C_VEL
LIN {X 0,Y 234.844,Z 729.64,A -85,B 0,C 180,E1 9119.316,E2 9119.316} C_VEL
LIN {X 0,Y 235.882,Z 728.515,A -85,B 0,C 180,E1 9118.804,E2 9118.804} C_VEL
LIN {X 0,Y 238.694,Z 727.842,A -85,B 0,C 180,E1 9118.144,E2 9118.144} C_VEL
LIN {X 0,Y 242.482,Z 724.499,A -85,B 0,C 180,E1 9117.429,E2 9117.429} C_VEL
LIN {X 0,Y 243.695,Z 723.279,A -85,B 0,C 180,E1 9117.213,E2 9117.213} C_VEL
LIN {X 0,Y 248.088,Z 733.108,A -85,B 0,C 180,E1 9115.906,E2 9115.906} C_VEL
LIN {X 0,Y 250.538,Z 752.544,A -85,B 0,C 180,E1 9114.68,E2 9114.68} C_VEL
LIN {X 0,Y 244.596,Z 860.643,A -85,B 0,C 180,E1 9111.713,E2 9111.713} C_VEL
LIN {X 0,Y 243.158,Z 878.302,A -85,B 0,C 180,E1 9110.86,E2 9110.86} C_VEL
LIN {X 0,Y 240.941,Z 895.037,A -85,B 0,C 180,E1 9109.642,E2 9109.642} C_VEL
LIN {X 0,Y 237.955,Z 911.676,A -85,B 0,C 180,E1 9107.99,E2 9107.99} C_VEL
LIN {X 0,Y 234.487,Z 927.181,A -85,B 0,C 180,E1 9105.964,E2 9105.964} C_VEL
LIN {X 0,Y 230.666,Z 941.521,A -85,B 0,C 180,E1 9103.538,E2 9103.538} C_VEL
LIN {X 0,Y 226.681,Z 954.843,A -85,B 0,C 180,E1 9100.677,E2 9100.677} C_VEL
LIN {X 0,Y 222.847,Z 966.634,A -85,B 0,C 180,E1 9097.477,E2 9097.477} C_VEL
LIN {X 0,Y 219.305,Z 976.895,A -85,B 0,C 180,E1 9093.922,E2 9093.922} C_VEL
LIN {X 0,Y 216.254,Z 985.729,A -85,B 0,C 180,E1 9090.001,E2 9090.001} C_VEL
LIN {X 0,Y 213.854,Z 993.11,A -85,B 0,C 180,E1 9085.711,E2 9085.711} C_VEL
LIN {X 0,Y 212.303,Z 998.618,A -85,B 0,C 180,E1 9081.333,E2 9081.333} C_VEL
LIN {X 0,Y 211.498,Z 1002.595,A -85,B 0,C 180,E1 9076.607,E2 9076.607} C_VEL
LIN {X 0,Y 211.54,Z 1004.837,A -85,B 0,C 180,E1 9071.815,E2 9071.815} C_VEL
LIN {X 0,Y 212.46,Z 1005.356,A -85,B 0,C 180,E1 9067.008,E2 9067.008} C_VEL
LIN {X 0,Y 214.368,Z 1004.027,A -85,B 0,C 180,E1 9062.198,E2 9062.198} C_VEL
LIN {X 0,Y 217.396,Z 1000.841,A -85,B 0,C 180,E1 9057.445,E2 9057.445} C_VEL
LIN {X 0,Y 221.352,Z 995.995,A -85,B 0,C 180,E1 9053.076,E2 9053.076} C_VEL
LIN {X 0,Y 226.033,Z 989.58,A -85,B 0,C 180,E1 9049.105,E2 9049.105} C_VEL
LIN {X 0,Y 231.63,Z 981.122,A -85,B 0,C 180,E1 9045.284,E2 9045.284} C_VEL
LIN {X 0,Y 237.641,Z 971.078,A -85,B 0,C 180,E1 9041.866,E2 9041.866} C_VEL
LIN {X 0,Y 243.742,Z 959.556,A -85,B 0,C 180,E1 9038.876,E2 9038.876} C_VEL
LIN {X 0,Y 249.538,Z 947.018,A -85,B 0,C 180,E1 9036.355,E2 9036.355} C_VEL
LIN {X 0,Y 255.024,Z 933.222,A -85,B 0,C 180,E1 9034.183,E2 9034.183} C_VEL
LIN {X 0,Y 259.896,Z 918.588,A -85,B 0,C 180,E1 9032.388,E2 9032.388} C_VEL
LIN {X 0,Y 264.162,Z 902.482,A -85,B 0,C 180,E1 9030.88,E2 9030.88} C_VEL
LIN {X 0,Y 267.487,Z 885.535,A -85,B 0,C 180,E1 9029.703,E2 9029.703} C_VEL
LIN {X 0,Y 269.764,Z 868.048,A -85,B 0,C 180,E1 9028.853,E2 9028.853} C_VEL
LIN {X 0,Y 271.62,Z 842.389,A -85,B 0,C 180,E1 9028.095,E2 9028.095} C_VEL
LIN {X 0,Y 271.62,Z 834.814,A -85,B 0,C 180,E1 9027.733,E2 9027.733} C_VEL
LIN {X 0,Y 269.665,Z 815.038,A -85,B 0,C 180,E1 9026.14,E2 9026.14} C_VEL
LIN {X 0,Y 269.767,Z 808.526,A -85,B 0,C 180,E1 9025.844,E2 9025.844} C_VEL
LIN {X 0,Y 273.117,Z 764.312,A -85,B 0,C 180,E1 9024.737,E2 9024.737} C_VEL
LIN {X 0,Y 268.275,Z 754.258,A -85,B 0,C 180,E1 9022.401,E2 9022.401} C_VEL
LIN {X 0,Y 262.802,Z 744.281,A -85,B 0,C 180,E1 9019.503,E2 9019.503} C_VEL
LIN {X 0,Y 259.242,Z 738.341,A -85,B 0,C 180,E1 9017.392,E2 9017.392} C_VEL
LIN {X 0,Y 255.757,Z 732.744,A -85,B 0,C 180,E1 9015.058,E2 9015.058} C_VEL
LIN {X 0,Y 252.788,Z 728.228,A -85,B 0,C 180,E1 9012.798,E2 9012.798} C_VEL
LIN {X 0,Y 248.428,Z 721.72,A -85,B 0,C 180,E1 9008.681,E2 9008.681} C_VEL
LIN {X 0,Y 244.934,Z 716.838,A -85,B 0,C 180,E1 9003.98,E2 9003.98} C_VEL
LIN {X 0,Y 242.614,Z 713.645,A -85,B 0,C 180,E1 8997.402,E2 8997.402} C_VEL
LIN {X 0,Y 242.922,Z 713.935,A -85,B 0,C 180,E1 8991.956,E2 8991.956} C_VEL
LIN {X 0,Y 246.1,Z 718.031,A -85,B 0,C 180,E1 8985.17,E2 8985.17} C_VEL
LIN {X 0,Y 247.884,Z 720.83,A -85,B 0,C 180,E1 8982.876,E2 8982.876} C_VEL
LIN {X 0,Y 251.14,Z 725.076,A -85,B 0,C 180,E1 8979.613,E2 8979.613} C_VEL
LIN {X 0,Y 256.266,Z 732.56,A -85,B 0,C 180,E1 8975.571,E2 8975.571} C_VEL
LIN {X 0,Y 261.242,Z 740.439,A -85,B 0,C 180,E1 8972.413,E2 8972.413} C_VEL
LIN {X 0,Y 265.378,Z 747.345,A -85,B 0,C 180,E1 8970.114,E2 8970.114} C_VEL
LIN {X 0,Y 270.562,Z 756.914,A -85,B 0,C 180,E1 8967.505,E2 8967.505} C_VEL
LIN {X 0,Y 273.8,Z 763.712,A -85,B 0,C 180,E1 8966.002,E2 8966.002} C_VEL
LIN {X 0,Y 273.142,Z 774.107,A -85,B 0,C 180,E1 8965.702,E2 8965.702} C_VEL
LIN {X 0,Y 263.778,Z 897.12,A -85,B 0,C 180,E1 8962.659,E2 8962.659} C_VEL
LIN {X 0,Y 260.935,Z 915.757,A -85,B 0,C 180,E1 8961.935,E2 8961.935} C_VEL
LIN {X 0,Y 256.854,Z 933.693,A -85,B 0,C 180,E1 8960.949,E2 8960.949} C_VEL
LIN {X 0,Y 251.501,Z 951.715,A -85,B 0,C 180,E1 8959.58,E2 8959.58} C_VEL
LIN {X 0,Y 245.775,Z 967.731,A -85,B 0,C 180,E1 8957.939,E2 8957.939} C_VEL
LIN {X 0,Y 239.478,Z 983.007,A -85,B 0,C 180,E1 8955.899,E2 8955.899} C_VEL
LIN {X 0,Y 232.786,Z 997.478,A -85,B 0,C 180,E1 8953.411,E2 8953.411} C_VEL
LIN {X 0,Y 225.709,Z 1011.533,A -85,B 0,C 180,E1 8950.297,E2 8950.297} C_VEL
LIN {X 0,Y 219.034,Z 1023.984,A -85,B 0,C 180,E1 8946.726,E2 8946.726} C_VEL
LIN {X 0,Y 213.04,Z 1034.998,A -85,B 0,C 180,E1 8942.664,E2 8942.664} C_VEL
LIN {X 0,Y 208.004,Z 1044.564,A -85,B 0,C 180,E1 8938.104,E2 8938.104} C_VEL
LIN {X 0,Y 204.149,Z 1052.767,A -85,B 0,C 180,E1 8932.962,E2 8932.962} C_VEL
LIN {X 0,Y 201.922,Z 1059.115,A -85,B 0,C 180,E1 8927.58,E2 8927.58} C_VEL
LIN {X 0,Y 201.243,Z 1063.443,A -85,B 0,C 180,E1 8922.335,E2 8922.335} C_VEL
LIN {X 0,Y 201.742,Z 1066.061,A -85,B 0,C 180,E1 8917.117,E2 8917.117} C_VEL
LIN {X 0,Y 202.624,Z 1066.902,A -85,B 0,C 180,E1 8912.545,E2 8912.545} C_VEL
LIN {X 0,Y 202.898,Z 1066.511,A -85,B 0,C 180,E1 8909.152,E2 8909.152} C_VEL
LIN {X 0,Y 202.411,Z 1064.86,A -85,B 0,C 180,E1 8905.182,E2 8905.182} C_VEL
LIN {X 0,Y 201.533,Z 1062.797,A -85,B 0,C 180,E1 8899.999,E2 8899.999} C_VEL
LIN {X 0,Y 201.537,Z 1059.281,A -85,B 0,C 180,E1 8895.335,E2 8895.335} C_VEL
LIN {X 0,Y 202.822,Z 1053.27,A -85,B 0,C 180,E1 8890.113,E2 8890.113} C_VEL
LIN {X 0,Y 205.466,Z 1045.518,A -85,B 0,C 180,E1 8885.259,E2 8885.259} C_VEL
LIN {X 0,Y 209.504,Z 1035.595,A -85,B 0,C 180,E1 8880.555,E2 8880.555} C_VEL
LIN {X 0,Y 214.238,Z 1024.745,A -85,B 0,C 180,E1 8876.583,E2 8876.583} C_VEL
LIN {X 0,Y 220.095,Z 1011.651,A -85,B 0,C 180,E1 8872.828,E2 8872.828} C_VEL
LIN {X 0,Y 226.017,Z 997.882,A -85,B 0,C 180,E1 8869.767,E2 8869.767} C_VEL
LIN {X 0,Y 232.085,Z 982.732,A -85,B 0,C 180,E1 8867.102,E2 8867.102} C_VEL
LIN {X 0,Y 237.935,Z 966.392,A -85,B 0,C 180,E1 8864.908,E2 8864.908} C_VEL
LIN {X 0,Y 242.985,Z 950.071,A -85,B 0,C 180,E1 8863.252,E2 8863.252} C_VEL
LIN {X 0,Y 247.416,Z 932.358,A -85,B 0,C 180,E1 8861.962,E2 8861.962} C_VEL
LIN {X 0,Y 251.006,Z 912.397,A -85,B 0,C 180,E1 8860.943,E2 8860.943} C_VEL
LIN {X 0,Y 269.775,Z 800.483,A -85,B 0,C 180,E1 8856.605,E2 8856.605} C_VEL
LIN {X 0,Y 274.466,Z 773.527,A -85,B 0,C 180,E1 8855.48,E2 8855.48} C_VEL
LIN {X 0,Y 275.861,Z 768.195,A -85,B 0,C 180,E1 8855.19,E2 8855.19} C_VEL
LIN {X 0,Y 279.109,Z 758.84,A -85,B 0,C 180,E1 8854.319,E2 8854.319} C_VEL
LIN {X 0,Y 280.494,Z 754.193,A -85,B 0,C 180,E1 8852.698,E2 8852.698} C_VEL
LIN {X 0,Y 279.337,Z 757.247,A -85,B 0,C 180,E1 8849.977,E2 8849.977} C_VEL
LIN {X 0,Y 278.375,Z 761.744,A -85,B 0,C 180,E1 8847.602,E2 8847.602} C_VEL
LIN {X 0,Y 278.599,Z 764.871,A -85,B 0,C 180,E1 8846.611,E2 8846.611} C_VEL
LIN {X 0,Y 278.174,Z 770.666,A -85,B 0,C 180,E1 8845.901,E2 8845.901} C_VEL
LIN {X 0,Y 262.828,Z 868.818,A -85,B 0,C 180,E1 8842.352,E2 8842.352} C_VEL
LIN {X 0,Y 258.696,Z 900.201,A -85,B 0,C 180,E1 8840.806,E2 8840.806} C_VEL
LIN {X 0,Y 255.913,Z 916.06,A -85,B 0,C 180,E1 8839.677,E2 8839.677} C_VEL
LIN {X 0,Y 251.947,Z 931.902,A -85,B 0,C 180,E1 8838.151,E2 8838.151} C_VEL
LIN {X 0,Y 247.274,Z 946.305,A -85,B 0,C 180,E1 8836.321,E2 8836.321} C_VEL
LIN {X 0,Y 241.928,Z 959.692,A -85,B 0,C 180,E1 8834.113,E2 8834.113} C_VEL
LIN {X 0,Y 236.553,Z 971.03,A -85,B 0,C 180,E1 8831.705,E2 8831.705} C_VEL
LIN {X 0,Y 231.022,Z 981.1,A -85,B 0,C 180,E1 8828.963,E2 8828.963} C_VEL
LIN {X 0,Y 225.035,Z 990.538,A -85,B 0,C 180,E1 8825.572,E2 8825.572} C_VEL
LIN {X 0,Y 219.778,Z 997.6,A -85,B 0,C 180,E1 8822.085,E2 8822.085} C_VEL
LIN {X 0,Y 214.896,Z 1003.279,A -85,B 0,C 180,E1 8818.133,E2 8818.133} C_VEL
LIN {X 0,Y 210.626,Z 1007.175,A -85,B 0,C 180,E1 8813.731,E2 8813.731} C_VEL
LIN {X 0,Y 207.511,Z 1009.006,A -85,B 0,C 180,E1 8809.407,E2 8809.407} C_VEL
LIN {X 0,Y 205.21,Z 1008.995,A -85,B 0,C 180,E1 8804.74,E2 8804.74} C_VEL
LIN {X 0,Y 203.902,Z 1007.115,A -85,B 0,C 180,E1 8800.223,E2 8800.223} C_VEL
LIN {X 0,Y 203.363,Z 1003.346,A -85,B 0,C 180,E1 8795.606,E2 8795.606} C_VEL
LIN {X 0,Y 203.525,Z 997.853,A -85,B 0,C 180,E1 8791.22,E2 8791.22} C_VEL
LIN {X 0,Y 204.305,Z 990.846,A -85,B 0,C 180,E1 8787.096,E2 8787.096} C_VEL
LIN {X 0,Y 205.734,Z 981.532,A -85,B 0,C 180,E1 8782.94,E2 8782.94} C_VEL
LIN {X 0,Y 207.5,Z 971.483,A -85,B 0,C 180,E1 8779.419,E2 8779.419} C_VEL
LIN {X 0,Y 209.805,Z 958.773,A -85,B 0,C 180,E1 8775.909,E2 8775.909} C_VEL
LIN {X 0,Y 212.184,Z 945.072,A -85,B 0,C 180,E1 8772.94,E2 8772.94} C_VEL
LIN {X 0,Y 214.405,Z 931.011,A -85,B 0,C 180,E1 8770.523,E2 8770.523} C_VEL
LIN {X 0,Y 216.625,Z 914.333,A -85,B 0,C 180,E1 8768.31,E2 8768.31} C_VEL
LIN {X 0,Y 218.341,Z 897.409,A -85,B 0,C 180,E1 8766.657,E2 8766.657} C_VEL
LIN {X 0,Y 219.502,Z 880.508,A -85,B 0,C 180,E1 8765.496,E2 8765.496} C_VEL
LIN {X 0,Y 222.109,Z 827.102,A -85,B 0,C 180,E1 8763.171,E2 8763.171} C_VEL
LIN {X 0,Y 227.235,Z 755.674,A -85,B 0,C 180,E1 8760.269,E2 8760.269} C_VEL
LIN {X 0,Y 228.474,Z 749.726,A -85,B 0,C 180,E1 8759.756,E2 8759.756} C_VEL
LIN {X 0,Y 231.334,Z 746.065,A -85,B 0,C 180,E1 8759.117,E2 8759.117} C_VEL
LIN {X 0,Y 234.236,Z 741.205,A -85,B 0,C 180,E1 8758.629,E2 8758.629} C_VEL
LIN {X 0,Y 235.961,Z 737.42,A -85,B 0,C 180,E1 8758.382,E2 8758.382} C_VEL
LIN {X 0,Y 236.869,Z 736.369,A -85,B 0,C 180,E1 8758.215,E2 8758.215} C_VEL
LIN {X 0,Y 240.927,Z 734.815,A -85,B 0,C 180,E1 8757.362,E2 8757.362} C_VEL
LIN {X 0,Y 241.614,Z 734.464,A -85,B 0,C 180,E1 8757.225,E2 8757.225} C_VEL
LIN {X 0,Y 242.459,Z 737.186,A -85,B 0,C 180,E1 8756.934,E2 8756.934} C_VEL
LIN {X 0,Y 244.437,Z 753.758,A -85,B 0,C 180,E1 8755.867,E2 8755.867} C_VEL
LIN {X 0,Y 238.282,Z 861.18,A -85,B 0,C 180,E1 8752.872,E2 8752.872} C_VEL
LIN {X 0,Y 236.778,Z 878.935,A -85,B 0,C 180,E1 8752.003,E2 8752.003} C_VEL
LIN {X 0,Y 234.412,Z 896.035,A -85,B 0,C 180,E1 8750.735,E2 8750.735} C_VEL
LIN {X 0,Y 231.299,Z 912.644,A -85,B 0,C 180,E1 8749.049,E2 8749.049} C_VEL
LIN {X 0,Y 227.681,Z 928.135,A -85,B 0,C 180,E1 8746.981,E2 8746.981} C_VEL
LIN {X 0,Y 223.693,Z 942.48,A -85,B 0,C 180,E1 8744.496,E2 8744.496} C_VEL
LIN {X 0,Y 219.525,Z 955.812,A -85,B 0,C 180,E1 8741.561,E2 8741.561} C_VEL
LIN {X 0,Y 215.51,Z 967.617,A -85,B 0,C 180,E1 8738.27,E2 8738.27} C_VEL
LIN {X 0,Y 211.794,Z 977.903,A -85,B 0,C 180,E1 8734.604,E2 8734.604} C_VEL
LIN {X 0,Y 208.586,Z 986.762,A -85,B 0,C 180,E1 8730.55,E2 8730.55} C_VEL
LIN {X 0,Y 206.058,Z 994.168,A -85,B 0,C 180,E1 8726.105,E2 8726.105} C_VEL
LIN {X 0,Y 204.422,Z 999.716,A -85,B 0,C 180,E1 8721.563,E2 8721.563} C_VEL
